KUKA KRL program: EPS_2_25694_GD05_A_20260114065905.src

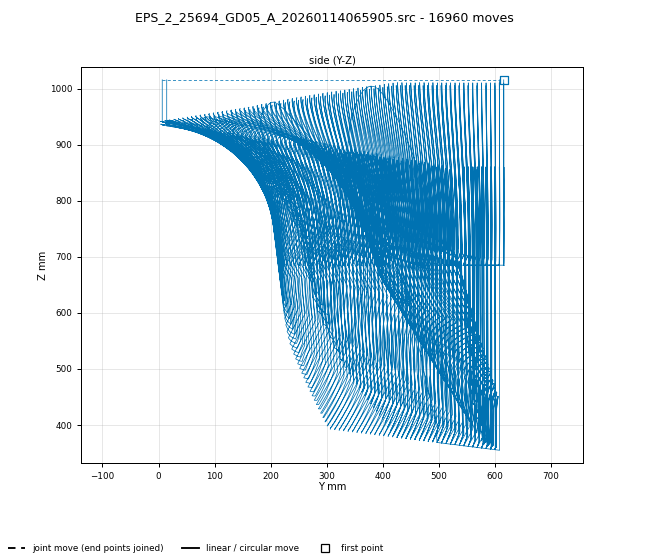
[picture p0: tool path of EPS_2_25694_GD05_A_20260114065905.src, 16960 of 16962 moves have a stored position in this frame; points joined in program order, loops and branches not executed]
&ACCESS RVP
&REL 4
&COMMENT QRS 19112012
&PARAM EDITMASK = *
DEF PART()
EXT BAS (BAS_COMMAND :IN,REAL :IN )
INT I
BAS (#INITMOV,0 )

;KUKA QRS Post kuka4.cps  Date:22-06-2017 !

File_ID=2971

QRS_PRE_INIT()

;Init var - Until changes are made in qrs_pre_init
Outlet_Square_prg=0
Inlet_1_Square_prg=0
Inlet_2_Square_prg=0
Inlet_3_Square_prg=0
Inlet_4_Square_prg=0
Inlet_5_Square_prg=0

Outlet_1={X 0.000, Y 425.000, Z 739.000, B 0.000, E1 0.000 }
Inlet_1={X 0.000, Y 500.470, Z 672.500, B 0.000, E1 180.000 }
Inlet_2={X 0.000, Y 520.810, Z 600.000, B 0.000, E1 270.000 }
Outlet_1_type=533
Inlet_1_type=366
Inlet_2_type=251
;QRS#1=Sidecore dimensions
;QRS#2=525-21" Concrete
;QRS#3=375-15" PVC SDR 35
;QRS#4=250-10" PVC SDR 35
;QRS#5=
;QRS#6=
;QRS#7=
;QRS#8=
;QRS#9=S306-32
;QRS#10=20Y PSX
;QRS#11=14M PSX
;QRS#12=
;QRS#13=
;QRS#14=
;QRS#15=
;QRS#16=1220x127x1372 4,5'
;QRS#17=EPS Height
;QRS#18=1005,5
;QRS#19=*
;QRS#20= UPDATED VERSION 22-06-2017
;QRS#21=*
Outlet_Square=0250
Inlet_1_Square=0250
Inlet_2_Square=0100
Inlet_3_Square=0
Inlet_4_Square=0
Inlet_5_Square=0
Mill_Square=1
Outlet_Square_Prg=263
Inlet_1_Square_prg=252
Inlet_2_Square_prg=205

QRS_INIT()

$ADVANCE=5

; T1
PTP {E1 172.561,E2 172.561}
PTP {X 0,Y 615.584,A -85,B 0,C 180,E1 172.561,E2 172.561,E3 0,E4 0,E5 0,E6 0}
QRS_SPEED_INIT()
LIN {X 0,Y 615.584,Z 1015.5,A -85,B 0,C 180,E1 172.561,E2 172.561,E3 0,E4 0,E5 0,E6 0} C_VEL
LIN {X 0,Y 615.584,Z 687.03,A -85,B 0,C 180,E1 172.561,E2 172.561} C_VEL
LIN {X 0,Y 615.53,Z 685.03,A -85,B 0,C 180,E1 172.747,E2 172.747} C_VEL
LIN {X 0,Y 615.824,Z 685.03,A -85,B 0,C 180,E1 176.52,E2 176.52} C_VEL
LIN {X 0,Y 615.876,Z 685.03,A -85,B 0,C 180,E1 181.159,E2 181.159} C_VEL
LIN {X 0,Y 615.817,Z 685.03,A -85,B 0,C 180,E1 185.807,E2 185.807} C_VEL
LIN {X 0,Y 615.791,Z 685.03,A -85,B 0,C 180,E1 190.494,E2 190.494} C_VEL
LIN {X 0,Y 615.808,Z 685.03,A -85,B 0,C 180,E1 195.252,E2 195.252} C_VEL
LIN {X 0,Y 615.745,Z 685.03,A -85,B 0,C 180,E1 200.123,E2 200.123} C_VEL
LIN {X 0,Y 615.743,Z 685.03,A -85,B 0,C 180,E1 205.15,E2 205.15} C_VEL
LIN {X 0,Y 615.401,Z 685.03,A -85,B 0,C 180,E1 209.459,E2 209.459} C_VEL
LIN {X 0,Y 615.733,Z 685.03,A -85,B 0,C 180,E1 210.395,E2 210.395} C_VEL
LIN {X 0,Y 615.144,Z 685.03,A -85,B 0,C 180,E1 213.844,E2 213.844} C_VEL
LIN {X 0,Y 615.689,Z 685.03,A -85,B 0,C 180,E1 215.941,E2 215.941} C_VEL
LIN {X 0,Y 615.421,Z 685.03,A -85,B 0,C 180,E1 217.844,E2 217.844} C_VEL
LIN {X 0,Y 615.368,Z 685.03,A -85,B 0,C 180,E1 218.885,E2 218.885} C_VEL
LIN {X 0,Y 615.634,Z 685.03,A -85,B 0,C 180,E1 221.502,E2 221.502} C_VEL
LIN {X 0,Y 615.674,Z 685.03,A -85,B 0,C 180,E1 225.105,E2 225.105} C_VEL
LIN {X 0,Y 615.272,Z 685.03,A -85,B 0,C 180,E1 228.536,E2 228.536} C_VEL
LIN {X 0,Y 615.659,Z 685.03,A -85,B 0,C 180,E1 231.137,E2 231.137} C_VEL
LIN {X 0,Y 615.631,Z 685.03,A -85,B 0,C 180,E1 236.089,E2 236.089} C_VEL
LIN {X 0,Y 615.749,Z 685.03,A -85,B 0,C 180,E1 236.879,E2 236.879} C_VEL
LIN {X 0,Y 615.824,Z 685.03,A -85,B 0,C 180,E1 240.42,E2 240.42} C_VEL
LIN {X 0,Y 615.203,Z 685.053,A -85,B 0,C 180,E1 240.571,E2 240.571} C_VEL
LIN {X 0,Y 615.421,Z 754.722,A -85,B 0,C 180,E1 241.502,E2 241.502} C_VEL
LIN {X 0,Y 615.517,Z 765.422,A -85,B 0,C 180,E1 241.682,E2 241.682} C_VEL
LIN {X 0,Y 615.533,Z 778.963,A -85,B 0,C 180,E1 241.97,E2 241.97} C_VEL
LIN {X 0,Y 615.511,Z 788.536,A -85,B 0,C 180,E1 242.211,E2 242.211} C_VEL
LIN {X 0,Y 615.673,Z 804.515,A -85,B 0,C 180,E1 242.705,E2 242.705} C_VEL
LIN {X 0,Y 615.632,Z 816.95,A -85,B 0,C 180,E1 243.151,E2 243.151} C_VEL
LIN {X 0,Y 615.564,Z 826.866,A -85,B 0,C 180,E1 243.554,E2 243.554} C_VEL
LIN {X 0,Y 615.704,Z 842.591,A -85,B 0,C 180,E1 244.286,E2 244.286} C_VEL
LIN {X 0,Y 615.691,Z 854.939,A -85,B 0,C 180,E1 244.935,E2 244.935} C_VEL
LIN {X 0,Y 615.678,Z 866.614,A -85,B 0,C 180,E1 245.617,E2 245.617} C_VEL
LIN {X 0,Y 615.714,Z 878.406,A -85,B 0,C 180,E1 246.379,E2 246.379} C_VEL
LIN {X 0,Y 615.719,Z 889.085,A -85,B 0,C 180,E1 247.135,E2 247.135} C_VEL
LIN {X 0,Y 615.705,Z 900.389,A -85,B 0,C 180,E1 248.011,E2 248.011} C_VEL
LIN {X 0,Y 615.703,Z 909.651,A -85,B 0,C 180,E1 248.791,E2 248.791} C_VEL
LIN {X 0,Y 615.752,Z 919.788,A -85,B 0,C 180,E1 249.723,E2 249.723} C_VEL
LIN {X 0,Y 615.721,Z 929.052,A -85,B 0,C 180,E1 250.646,E2 250.646} C_VEL
LIN {X 0,Y 615.678,Z 937.422,A -85,B 0,C 180,E1 251.549,E2 251.549} C_VEL
LIN {X 0,Y 615.759,Z 945.774,A -85,B 0,C 180,E1 252.531,E2 252.531} C_VEL
LIN {X 0,Y 615.711,Z 953.68,A -85,B 0,C 180,E1 253.541,E2 253.541} C_VEL
LIN {X 0,Y 615.577,Z 960.425,A -85,B 0,C 180,E1 254.472,E2 254.472} C_VEL
LIN {X 0,Y 615.67,Z 968.06,A -85,B 0,C 180,E1 255.644,E2 255.644} C_VEL
LIN {X 0,Y 615.808,Z 973.436,A -85,B 0,C 180,E1 256.543,E2 256.543} C_VEL
LIN {X 0,Y 615.572,Z 979.909,A -85,B 0,C 180,E1 257.728,E2 257.728} C_VEL
LIN {X 0,Y 615.608,Z 985.624,A -85,B 0,C 180,E1 258.913,E2 258.913} C_VEL
LIN {X 0,Y 615.819,Z 990.635,A -85,B 0,C 180,E1 260.096,E2 260.096} C_VEL
LIN {X 0,Y 615.602,Z 995.063,A -85,B 0,C 180,E1 261.268,E2 261.268} C_VEL
LIN {X 0,Y 615.662,Z 999.448,A -85,B 0,C 180,E1 262.653,E2 262.653} C_VEL
LIN {X 0,Y 615.802,Z 1002.362,A -85,B 0,C 180,E1 263.747,E2 263.747} C_VEL
LIN {X 0,Y 615.601,Z 1004.4,A -85,B 0,C 180,E1 264.657,E2 264.657} C_VEL
LIN {X 0,Y 615.536,Z 1006.161,A -85,B 0,C 180,E1 265.588,E2 265.588} C_VEL
LIN {X 0,Y 615.635,Z 1007.593,A -85,B 0,C 180,E1 266.519,E2 266.519} C_VEL
LIN {X 0,Y 615.7,Z 1009.056,A -85,B 0,C 180,E1 267.912,E2 267.912} C_VEL
LIN {X 0,Y 615.544,Z 1009.716,A -85,B 0,C 180,E1 268.84,E2 268.84} C_VEL
LIN {X 0,Y 615.842,Z 1009.659,A -85,B 0,C 180,E1 271.16,E2 271.16} C_VEL
LIN {X 0,Y 615.558,Z 1008.719,A -85,B 0,C 180,E1 272.553,E2 272.553} C_VEL
LIN {X 0,Y 615.598,Z 1006.935,A -85,B 0,C 180,E1 273.947,E2 273.947} C_VEL
LIN {X 0,Y 615.805,Z 1005.333,A -85,B 0,C 180,E1 274.876,E2 274.876} C_VEL
LIN {X 0,Y 615.605,Z 1002.404,A -85,B 0,C 180,E1 276.252,E2 276.252} C_VEL
LIN {X 0,Y 615.625,Z 999.258,A -85,B 0,C 180,E1 277.421,E2 277.421} C_VEL
LIN {X 0,Y 615.798,Z 995.032,A -85,B 0,C 180,E1 278.73,E2 278.73} C_VEL
LIN {X 0,Y 615.583,Z 990.668,A -85,B 0,C 180,E1 279.908,E2 279.908} C_VEL
LIN {X 0,Y 615.638,Z 985.619,A -85,B 0,C 180,E1 281.087,E2 281.087} C_VEL
LIN {X 0,Y 615.808,Z 979.88,A -85,B 0,C 180,E1 282.268,E2 282.268} C_VEL
LIN {X 0,Y 615.627,Z 973.452,A -85,B 0,C 180,E1 283.461,E2 283.461} C_VEL
LIN {X 0,Y 615.697,Z 966.191,A -85,B 0,C 180,E1 284.655,E2 284.655} C_VEL
LIN {X 0,Y 615.81,Z 960.633,A -85,B 0,C 180,E1 285.488,E2 285.488} C_VEL
LIN {X 0,Y 615.662,Z 951.196,A -85,B 0,C 180,E1 286.791,E2 286.791} C_VEL
LIN {X 0,Y 615.737,Z 942.603,A -85,B 0,C 180,E1 287.853,E2 287.853} C_VEL
LIN {X 0,Y 615.77,Z 934.408,A -85,B 0,C 180,E1 288.785,E2 288.785} C_VEL
LIN {X 0,Y 615.695,Z 924.518,A -85,B 0,C 180,E1 289.817,E2 289.817} C_VEL
LIN {X 0,Y 615.712,Z 916.531,A -85,B 0,C 180,E1 290.588,E2 290.588} C_VEL
LIN {X 0,Y 615.743,Z 906.028,A -85,B 0,C 180,E1 291.519,E2 291.519} C_VEL
LIN {X 0,Y 615.702,Z 896.055,A -85,B 0,C 180,E1 292.335,E2 292.335} C_VEL
LIN {X 0,Y 615.701,Z 886.287,A -85,B 0,C 180,E1 293.072,E2 293.072} C_VEL
LIN {X 0,Y 615.683,Z 874.63,A -85,B 0,C 180,E1 293.874,E2 293.874} C_VEL
LIN {X 0,Y 615.702,Z 862.594,A -85,B 0,C 180,E1 294.623,E2 294.623} C_VEL
LIN {X 0,Y 615.65,Z 851.876,A -85,B 0,C 180,E1 295.235,E2 295.235} C_VEL
LIN {X 0,Y 615.643,Z 841.007,A -85,B 0,C 180,E1 295.797,E2 295.797} C_VEL
LIN {X 0,Y 615.687,Z 826.859,A -85,B 0,C 180,E1 296.441,E2 296.441} C_VEL
LIN {X 0,Y 615.612,Z 813.654,A -85,B 0,C 180,E1 296.972,E2 296.972} C_VEL
LIN {X 0,Y 615.555,Z 804.507,A -85,B 0,C 180,E1 297.301,E2 297.301} C_VEL
LIN {X 0,Y 615.62,Z 787.838,A -85,B 0,C 180,E1 297.801,E2 297.801} C_VEL
LIN {X 0,Y 615.469,Z 776.068,A -85,B 0,C 180,E1 298.103,E2 298.103} C_VEL
LIN {X 0,Y 615.637,Z 761.901,A -85,B 0,C 180,E1 298.376,E2 298.376} C_VEL
LIN {X 0,Y 615.601,Z 741.63,A -85,B 0,C 180,E1 298.669,E2 298.669} C_VEL
LIN {X 0,Y 615.253,Z 685.03,A -85,B 0,C 180,E1 299.434,E2 299.434} C_VEL
LIN {X 0,Y 615.616,Z 685.03,A -85,B 0,C 180,E1 299.501,E2 299.501} C_VEL
LIN {X 0,Y 615.665,Z 685.03,A -85,B 0,C 180,E1 300.399,E2 300.399} C_VEL
LIN {X 0,Y 615.751,Z 685.03,A -85,B 0,C 180,E1 303.122,E2 303.122} C_VEL
LIN {X 0,Y 615.639,Z 685.03,A -85,B 0,C 180,E1 303.912,E2 303.912} C_VEL
LIN {X 0,Y 615.658,Z 685.03,A -85,B 0,C 180,E1 308.863,E2 308.863} C_VEL
LIN {X 0,Y 615.255,Z 685.03,A -85,B 0,C 180,E1 311.942,E2 311.942} C_VEL
LIN {X 0,Y 615.672,Z 685.03,A -85,B 0,C 180,E1 314.894,E2 314.894} C_VEL
LIN {X 0,Y 615.654,Z 685.03,A -85,B 0,C 180,E1 318.496,E2 318.496} C_VEL
LIN {X 0,Y 615.381,Z 685.03,A -85,B 0,C 180,E1 321.116,E2 321.116} C_VEL
LIN {X 0,Y 615.438,Z 685.03,A -85,B 0,C 180,E1 322.155,E2 322.155} C_VEL
LIN {X 0,Y 615.695,Z 685.03,A -85,B 0,C 180,E1 324.059,E2 324.059} C_VEL
LIN {X 0,Y 615.138,Z 685.03,A -85,B 0,C 180,E1 326.841,E2 326.841} C_VEL
LIN {X 0,Y 615.715,Z 685.03,A -85,B 0,C 180,E1 329.604,E2 329.604} C_VEL
LIN {X 0,Y 615.214,Z 685.03,A -85,B 0,C 180,E1 332.233,E2 332.233} C_VEL
LIN {X 0,Y 615.76,Z 685.03,A -85,B 0,C 180,E1 334.85,E2 334.85} C_VEL
LIN {X 0,Y 615.776,Z 685.03,A -85,B 0,C 180,E1 339.878,E2 339.878} C_VEL
LIN {X 0,Y 615.756,Z 685.03,A -85,B 0,C 180,E1 344.747,E2 344.747} C_VEL
LIN {X 0,Y 615.177,Z 685.03,A -85,B 0,C 180,E1 344.957,E2 344.957} C_VEL
LIN {X 0,Y 615.457,Z 685.827,A -85,B 0,C 180,E1 344.981,E2 344.981} C_VEL
LIN {X 0,Y 615.716,Z 687.593,A -85,B 0,C 180,E1 345.008,E2 345.008} C_VEL
LIN {X 0,Y 615.804,Z 728.118,A -85,B 0,C 180,E1 345.498,E2 345.498} C_VEL
LIN {X 0,Y 615.783,Z 737.858,A -85,B 0,C 180,E1 345.666,E2 345.666} C_VEL
LIN {X 0,Y 615.759,Z 747.806,A -85,B 0,C 180,E1 345.908,E2 345.908} C_VEL
LIN {X 0,Y 615.82,Z 756.4,A -85,B 0,C 180,E1 346.171,E2 346.171} C_VEL
LIN {X 0,Y 615.832,Z 766.418,A -85,B 0,C 180,E1 346.544,E2 346.544} C_VEL
LIN {X 0,Y 615.818,Z 774.745,A -85,B 0,C 180,E1 346.916,E2 346.916} C_VEL
LIN {X 0,Y 615.831,Z 783.402,A -85,B 0,C 180,E1 347.362,E2 347.362} C_VEL
LIN {X 0,Y 615.825,Z 792.017,A -85,B 0,C 180,E1 347.881,E2 347.881} C_VEL
LIN {X 0,Y 615.821,Z 799.559,A -85,B 0,C 180,E1 348.399,E2 348.399} C_VEL
LIN {X 0,Y 615.811,Z 808.029,A -85,B 0,C 180,E1 349.064,E2 349.064} C_VEL
LIN {X 0,Y 615.849,Z 814.611,A -85,B 0,C 180,E1 349.655,E2 349.655} C_VEL
LIN {X 0,Y 615.797,Z 821.882,A -85,B 0,C 180,E1 350.39,E2 350.39} C_VEL
LIN {X 0,Y 615.799,Z 828.194,A -85,B 0,C 180,E1 351.124,E2 351.124} C_VEL
LIN {X 0,Y 615.843,Z 833.772,A -85,B 0,C 180,E1 351.857,E2 351.857} C_VEL
LIN {X 0,Y 615.769,Z 838.545,A -85,B 0,C 180,E1 352.576,E2 352.576} C_VEL
LIN {X 0,Y 615.759,Z 842.466,A -85,B 0,C 180,E1 353.245,E2 353.245} C_VEL
LIN {X 0,Y 615.84,Z 847.264,A -85,B 0,C 180,E1 354.193,E2 354.193} C_VEL
LIN {X 0,Y 615.718,Z 851.122,A -85,B 0,C 180,E1 355.124,E2 355.124} C_VEL
LIN {X 0,Y 615.753,Z 854.265,A -85,B 0,C 180,E1 356.054,E2 356.054} C_VEL
LIN {X 0,Y 615.82,Z 856.63,A -85,B 0,C 180,E1 356.984,E2 356.984} C_VEL
LIN {X 0,Y 615.759,Z 857.615,A -85,B 0,C 180,E1 357.448,E2 357.448} C_VEL
LIN {X 0,Y 615.72,Z 858.999,A -85,B 0,C 180,E1 358.376,E2 358.376} C_VEL
LIN {X 0,Y 615.841,Z 859.769,A -85,B 0,C 180,E1 359.304,E2 359.304} C_VEL
LIN {X 0,Y 615.711,Z 859.892,A -85,B 0,C 180,E1 360.232,E2 360.232} C_VEL
LIN {X 0,Y 615.685,Z 859.413,A -85,B 0,C 180,E1 361.16,E2 361.16} C_VEL
LIN {X 0,Y 615.732,Z 858.891,A -85,B 0,C 180,E1 361.624,E2 361.624} C_VEL
LIN {X 0,Y 615.833,Z 857.437,A -85,B 0,C 180,E1 362.551,E2 362.551} C_VEL
LIN {X 0,Y 615.722,Z 855.292,A -85,B 0,C 180,E1 363.481,E2 363.481} C_VEL
LIN {X 0,Y 615.773,Z 852.487,A -85,B 0,C 180,E1 364.41,E2 364.41} C_VEL
LIN {X 0,Y 615.847,Z 850.762,A -85,B 0,C 180,E1 364.875,E2 364.875} C_VEL
LIN {X 0,Y 615.751,Z 846.849,A -85,B 0,C 180,E1 365.808,E2 365.808} C_VEL
LIN {X 0,Y 615.738,Z 841.761,A -85,B 0,C 180,E1 366.794,E2 366.794} C_VEL
LIN {X 0,Y 615.85,Z 836.822,A -85,B 0,C 180,E1 367.602,E2 367.602} C_VEL
LIN {X 0,Y 615.766,Z 830.942,A -85,B 0,C 180,E1 368.437,E2 368.437} C_VEL
LIN {X 0,Y 615.764,Z 825.022,A -85,B 0,C 180,E1 369.17,E2 369.17} C_VEL
LIN {X 0,Y 615.833,Z 819.636,A -85,B 0,C 180,E1 369.757,E2 369.757} C_VEL
LIN {X 0,Y 615.834,Z 813.655,A -85,B 0,C 180,E1 370.346,E2 370.346} C_VEL
LIN {X 0,Y 615.806,Z 806.983,A -85,B 0,C 180,E1 370.936,E2 370.936} C_VEL
LIN {X 0,Y 615.829,Z 799.335,A -85,B 0,C 180,E1 371.527,E2 371.527} C_VEL
LIN {X 0,Y 615.844,Z 791.773,A -85,B 0,C 180,E1 372.044,E2 372.044} C_VEL
LIN {X 0,Y 615.819,Z 783.109,A -85,B 0,C 180,E1 372.564,E2 372.564} C_VEL
LIN {X 0,Y 615.806,Z 774.421,A -85,B 0,C 180,E1 373.01,E2 373.01} C_VEL
LIN {X 0,Y 615.823,Z 766.055,A -85,B 0,C 180,E1 373.382,E2 373.382} C_VEL
LIN {X 0,Y 615.826,Z 755.927,A -85,B 0,C 180,E1 373.755,E2 373.755} C_VEL
LIN {X 0,Y 615.788,Z 747.254,A -85,B 0,C 180,E1 374.017,E2 374.017} C_VEL
LIN {X 0,Y 615.813,Z 739.659,A -85,B 0,C 180,E1 374.203,E2 374.203} C_VEL
LIN {X 0,Y 615.835,Z 729.706,A -85,B 0,C 180,E1 374.389,E2 374.389} C_VEL
LIN {X 0,Y 615.679,Z 699.013,A -85,B 0,C 180,E1 374.768,E2 374.768} C_VEL
LIN {X 0,Y 615.543,Z 686.33,A -85,B 0,C 180,E1 374.921,E2 374.921} C_VEL
LIN {X 0,Y 615.607,Z 685.03,A -85,B 0,C 180,E1 374.957,E2 374.957} C_VEL
LIN {X 0,Y 615.792,Z 685.03,A -85,B 0,C 180,E1 375.252,E2 375.252} C_VEL
LIN {X 0,Y 615.768,Z 685.03,A -85,B 0,C 180,E1 380.123,E2 380.123} C_VEL
LIN {X 0,Y 615.761,Z 685.03,A -85,B 0,C 180,E1 385.15,E2 385.15} C_VEL
LIN {X 0,Y 615.378,Z 685.03,A -85,B 0,C 180,E1 389.454,E2 389.454} C_VEL
LIN {X 0,Y 615.701,Z 685.03,A -85,B 0,C 180,E1 390.397,E2 390.397} C_VEL
LIN {X 0,Y 615.132,Z 685.03,A -85,B 0,C 180,E1 393.842,E2 393.842} C_VEL
LIN {X 0,Y 615.69,Z 685.03,A -85,B 0,C 180,E1 395.941,E2 395.941} C_VEL
LIN {X 0,Y 615.638,Z 685.03,A -85,B 0,C 180,E1 397.869,E2 397.869} C_VEL
LIN {X 0,Y 615.724,Z 685.03,A -85,B 0,C 180,E1 398.858,E2 398.858} C_VEL
LIN {X 0,Y 615.234,Z 685.03,A -85,B 0,C 180,E1 401.944,E2 401.944} C_VEL
LIN {X 0,Y 615.676,Z 685.03,A -85,B 0,C 180,E1 404.895,E2 404.895} C_VEL
LIN {X 0,Y 615.651,Z 685.03,A -85,B 0,C 180,E1 408.497,E2 408.497} C_VEL
LIN {X 0,Y 615.347,Z 685.03,A -85,B 0,C 180,E1 411.113,E2 411.113} C_VEL
LIN {X 0,Y 615.387,Z 685.03,A -85,B 0,C 180,E1 412.161,E2 412.161} C_VEL
LIN {X 0,Y 615.636,Z 685.03,A -85,B 0,C 180,E1 414.055,E2 414.055} C_VEL
LIN {X 0,Y 615.128,Z 685.03,A -85,B 0,C 180,E1 416.84,E2 416.84} C_VEL
LIN {X 0,Y 615.747,Z 685.03,A -85,B 0,C 180,E1 419.606,E2 419.606} C_VEL
LIN {X 0,Y 615.236,Z 685.03,A -85,B 0,C 180,E1 422.234,E2 422.234} C_VEL
LIN {X 0,Y 615.77,Z 685.03,A -85,B 0,C 180,E1 424.851,E2 424.851} C_VEL
LIN {X 0,Y 615.275,Z 685.03,A -85,B 0,C 180,E1 427.368,E2 427.368} C_VEL
LIN {X 0,Y 615.552,Z 685.03,A -85,B 0,C 180,E1 429.87,E2 429.87} C_VEL
LIN {X 0,Y 614.862,Z 685.03,A -85,B 0,C 180,E1 430.001,E2 430.001} C_VEL
LIN {X 0,Y 615.158,Z 686.38,A -85,B 0,C 180,E1 430.056,E2 430.056} C_VEL
LIN {X 0,Y 615.519,Z 688.076,A -85,B 0,C 180,E1 430.1,E2 430.1} C_VEL
LIN {X 0,Y 615.754,Z 695.441,A -85,B 0,C 180,E1 430.262,E2 430.262} C_VEL
LIN {X 0,Y 615.807,Z 705.296,A -85,B 0,C 180,E1 430.514,E2 430.514} C_VEL
LIN {X 0,Y 615.785,Z 714.797,A -85,B 0,C 180,E1 430.801,E2 430.801} C_VEL
LIN {X 0,Y 615.726,Z 723.53,A -85,B 0,C 180,E1 431.106,E2 431.106} C_VEL
LIN {X 0,Y 615.788,Z 732.709,A -85,B 0,C 180,E1 431.477,E2 431.477} C_VEL
LIN {X 0,Y 615.779,Z 741.924,A -85,B 0,C 180,E1 431.897,E2 431.897} C_VEL
LIN {X 0,Y 615.726,Z 750.371,A -85,B 0,C 180,E1 432.327,E2 432.327} C_VEL
LIN {X 0,Y 615.768,Z 758.249,A -85,B 0,C 180,E1 432.773,E2 432.773} C_VEL
LIN {X 0,Y 615.772,Z 765.444,A -85,B 0,C 180,E1 433.217,E2 433.217} C_VEL
LIN {X 0,Y 615.802,Z 774.115,A -85,B 0,C 180,E1 433.81,E2 433.81} C_VEL
LIN {X 0,Y 615.788,Z 781.849,A -85,B 0,C 180,E1 434.39,E2 434.39} C_VEL
LIN {X 0,Y 615.765,Z 789.814,A -85,B 0,C 180,E1 435.047,E2 435.047} C_VEL
LIN {X 0,Y 615.775,Z 796.45,A -85,B 0,C 180,E1 435.647,E2 435.647} C_VEL
LIN {X 0,Y 615.829,Z 803.981,A -85,B 0,C 180,E1 436.395,E2 436.395} C_VEL
LIN {X 0,Y 615.772,Z 809.484,A -85,B 0,C 180,E1 436.989,E2 436.989} C_VEL
LIN {X 0,Y 615.717,Z 815.784,A -85,B 0,C 180,E1 437.731,E2 437.731} C_VEL
LIN {X 0,Y 615.762,Z 821.496,A -85,B 0,C 180,E1 438.472,E2 438.472} C_VEL
LIN {X 0,Y 615.83,Z 826.677,A -85,B 0,C 180,E1 439.212,E2 439.212} C_VEL
LIN {X 0,Y 615.701,Z 832.297,A -85,B 0,C 180,E1 440.094,E2 440.094} C_VEL
LIN {X 0,Y 615.677,Z 835.681,A -85,B 0,C 180,E1 440.681,E2 440.681} C_VEL
LIN {X 0,Y 615.761,Z 840.253,A -85,B 0,C 180,E1 441.563,E2 441.563} C_VEL
LIN {X 0,Y 615.825,Z 843.092,A -85,B 0,C 180,E1 442.165,E2 442.165} C_VEL
LIN {X 0,Y 615.696,Z 846.093,A -85,B 0,C 180,E1 442.859,E2 442.859} C_VEL
LIN {X 0,Y 615.628,Z 849.335,A -85,B 0,C 180,E1 443.719,E2 443.719} C_VEL
LIN {X 0,Y 615.712,Z 852.329,A -85,B 0,C 180,E1 444.658,E2 444.658} C_VEL
LIN {X 0,Y 615.79,Z 854.78,A -85,B 0,C 180,E1 445.59,E2 445.59} C_VEL
LIN {X 0,Y 615.639,Z 856.773,A -85,B 0,C 180,E1 446.519,E2 446.519} C_VEL
LIN {X 0,Y 615.653,Z 858.252,A -85,B 0,C 180,E1 447.448,E2 447.448} C_VEL
LIN {X 0,Y 615.775,Z 859.568,A -85,B 0,C 180,E1 448.84,E2 448.84} C_VEL
LIN {X 0,Y 615.634,Z 859.928,A -85,B 0,C 180,E1 449.768,E2 449.768} C_VEL
LIN {X 0,Y 615.624,Z 859.908,A -85,B 0,C 180,E1 450.232,E2 450.232} C_VEL
LIN {X 0,Y 615.725,Z 859.514,A -85,B 0,C 180,E1 451.16,E2 451.16} C_VEL
LIN {X 0,Y 615.786,Z 858.668,A -85,B 0,C 180,E1 452.087,E2 452.087} C_VEL
LIN {X 0,Y 615.702,Z 858.137,A -85,B 0,C 180,E1 452.552,E2 452.552} C_VEL
LIN {X 0,Y 615.627,Z 856.622,A -85,B 0,C 180,E1 453.481,E2 453.481} C_VEL
LIN {X 0,Y 615.721,Z 854.584,A -85,B 0,C 180,E1 454.411,E2 454.411} C_VEL
LIN {X 0,Y 615.769,Z 852.048,A -85,B 0,C 180,E1 455.341,E2 455.341} C_VEL
LIN {X 0,Y 615.671,Z 848.986,A -85,B 0,C 180,E1 456.283,E2 456.283} C_VEL
LIN {X 0,Y 615.764,Z 844.496,A -85,B 0,C 180,E1 457.42,E2 457.42} C_VEL
LIN {X 0,Y 615.808,Z 841.234,A -85,B 0,C 180,E1 458.143,E2 458.143} C_VEL
LIN {X 0,Y 615.717,Z 838.386,A -85,B 0,C 180,E1 458.731,E2 458.731} C_VEL
LIN {X 0,Y 615.682,Z 833.542,A -85,B 0,C 180,E1 459.612,E2 459.612} C_VEL
LIN {X 0,Y 615.79,Z 828.06,A -85,B 0,C 180,E1 460.494,E2 460.494} C_VEL
LIN {X 0,Y 615.811,Z 823.014,A -85,B 0,C 180,E1 461.231,E2 461.231} C_VEL
LIN {X 0,Y 615.725,Z 817.46,A -85,B 0,C 180,E1 461.972,E2 461.972} C_VEL
LIN {X 0,Y 615.74,Z 811.326,A -85,B 0,C 180,E1 462.714,E2 462.714} C_VEL
LIN {X 0,Y 615.83,Z 804.554,A -85,B 0,C 180,E1 463.456,E2 463.456} C_VEL
LIN {X 0,Y 615.807,Z 798.651,A -85,B 0,C 180,E1 464.053,E2 464.053} C_VEL
LIN {X 0,Y 615.764,Z 792.222,A -85,B 0,C 180,E1 464.653,E2 464.653} C_VEL
LIN {X 0,Y 615.786,Z 785.195,A -85,B 0,C 180,E1 465.252,E2 465.252} C_VEL
LIN {X 0,Y 615.795,Z 777.438,A -85,B 0,C 180,E1 465.857,E2 465.857} C_VEL
LIN {X 0,Y 615.796,Z 770.063,A -85,B 0,C 180,E1 466.384,E2 466.384} C_VEL
LIN {X 0,Y 615.768,Z 762.769,A -85,B 0,C 180,E1 466.863,E2 466.863} C_VEL
LIN {X 0,Y 615.76,Z 754.276,A -85,B 0,C 180,E1 467.368,E2 467.368} C_VEL
LIN {X 0,Y 615.734,Z 744.638,A -85,B 0,C 180,E1 467.881,E2 467.881} C_VEL
LIN {X 0,Y 615.774,Z 735.788,A -85,B 0,C 180,E1 468.299,E2 468.299} C_VEL
LIN {X 0,Y 615.768,Z 726.909,A -85,B 0,C 180,E1 468.672,E2 468.672} C_VEL
LIN {X 0,Y 615.7,Z 718.531,A -85,B 0,C 180,E1 468.987,E2 468.987} C_VEL
LIN {X 0,Y 615.806,Z 708.175,A -85,B 0,C 180,E1 469.314,E2 469.314} C_VEL
LIN {X 0,Y 615.799,Z 698.822,A -85,B 0,C 180,E1 469.566,E2 469.566} C_VEL
LIN {X 0,Y 615.703,Z 688.908,A -85,B 0,C 180,E1 469.788,E2 469.788} C_VEL
LIN {X 0,Y 615.636,Z 685.03,A -85,B 0,C 180,E1 469.874,E2 469.874} C_VEL
LIN {X 0,Y 615.853,Z 685.03,A -85,B 0,C 180,E1 469.985,E2 469.985} C_VEL
LIN {X 0,Y 615.83,Z 685.03,A -85,B 0,C 180,E1 472.61,E2 472.61} C_VEL
LIN {X 0,Y 615.75,Z 685.03,A -85,B 0,C 180,E1 477.74,E2 477.74} C_VEL
LIN {X 0,Y 615.174,Z 685.03,A -85,B 0,C 180,E1 480.425,E2 480.425} C_VEL
LIN {X 0,Y 615.698,Z 685.03,A -85,B 0,C 180,E1 483.125,E2 483.125} C_VEL
LIN {X 0,Y 615.634,Z 685.03,A -85,B 0,C 180,E1 483.911,E2 483.911} C_VEL
LIN {X 0,Y 615.656,Z 685.03,A -85,B 0,C 180,E1 488.863,E2 488.863} C_VEL
LIN {X 0,Y 615.247,Z 685.03,A -85,B 0,C 180,E1 491.943,E2 491.943} C_VEL
LIN {X 0,Y 615.653,Z 685.03,A -85,B 0,C 180,E1 494.893,E2 494.893} C_VEL
LIN {X 0,Y 615.627,Z 685.03,A -85,B 0,C 180,E1 498.499,E2 498.499} C_VEL
LIN {X 0,Y 615.365,Z 685.03,A -85,B 0,C 180,E1 501.115,E2 501.115} C_VEL
LIN {X 0,Y 615.417,Z 685.03,A -85,B 0,C 180,E1 502.157,E2 502.157} C_VEL
LIN {X 0,Y 615.697,Z 685.03,A -85,B 0,C 180,E1 504.06,E2 504.06} C_VEL
LIN {X 0,Y 615.157,Z 685.03,A -85,B 0,C 180,E1 506.842,E2 506.842} C_VEL
LIN {X 0,Y 615.745,Z 685.03,A -85,B 0,C 180,E1 509.606,E2 509.606} C_VEL
LIN {X 0,Y 615.215,Z 685.03,A -85,B 0,C 180,E1 512.233,E2 512.233} C_VEL
LIN {X 0,Y 615.723,Z 685.03,A -85,B 0,C 180,E1 514.849,E2 514.849} C_VEL
LIN {X 0,Y 615.778,Z 685.03,A -85,B 0,C 180,E1 519.878,E2 519.878} C_VEL
LIN {X 0,Y 615.515,Z 685.03,A -85,B 0,C 180,E1 522.321,E2 522.321} C_VEL
LIN {X 0,Y 615.64,Z 685.03,A -85,B 0,C 180,E1 524.744,E2 524.744} C_VEL
LIN {X 0,Y 615.831,Z 685.03,A -85,B 0,C 180,E1 527.139,E2 527.139} C_VEL
LIN {X 0,Y 615.834,Z 685.03,A -85,B 0,C 180,E1 531.857,E2 531.857} C_VEL
LIN {X 0,Y 615.53,Z 685.03,A -85,B 0,C 180,E1 532.747,E2 532.747} C_VEL
LIN {X 0,Y 611.514,Z 685.03,A -85,B 0,C 180,E1 534.334,E2 534.334} C_VEL
LIN {X 0,Y 607.65,Z 685.03,A -85,B 0,C 180,E1 535.941,E2 535.941} C_VEL
LIN {X 0,Y 607.884,Z 685.03,A -85,B 0,C 180,E1 541.425,E2 541.425} C_VEL
LIN {X 0,Y 607.635,Z 685.03,A -85,B 0,C 180,E1 546.599,E2 546.599} C_VEL
LIN {X 0,Y 607.552,Z 685.03,A -85,B 0,C 180,E1 551.463,E2 551.463} C_VEL
LIN {X 0,Y 607.655,Z 685.03,A -85,B 0,C 180,E1 555.855,E2 555.855} C_VEL
LIN {X 0,Y 607.757,Z 685.03,A -85,B 0,C 180,E1 560.343,E2 560.343} C_VEL
LIN {X 0,Y 607.766,Z 685.03,A -85,B 0,C 180,E1 564.968,E2 564.968} C_VEL
LIN {X 0,Y 607.612,Z 685.03,A -85,B 0,C 180,E1 569.783,E2 569.783} C_VEL
LIN {X 0,Y 607.625,Z 685.03,A -85,B 0,C 180,E1 576.586,E2 576.586} C_VEL
LIN {X 0,Y 607.595,Z 685.03,A -85,B 0,C 180,E1 582.11,E2 582.11} C_VEL
LIN {X 0,Y 607.278,Z 685.03,A -85,B 0,C 180,E1 587.863,E2 587.863} C_VEL
LIN {X 0,Y 607.283,Z 685.03,A -85,B 0,C 180,E1 592.668,E2 592.668} C_VEL
LIN {X 0,Y 607.689,Z 685.03,A -85,B 0,C 180,E1 597.593,E2 597.593} C_VEL
LIN {X 0,Y 607.848,Z 685.03,A -85,B 0,C 180,E1 600.149,E2 600.149} C_VEL
LIN {X 0,Y 608.576,Z 775.688,A -85,B 0,C 180,E1 601.541,E2 601.541} C_VEL
LIN {X 0,Y 608.525,Z 816.222,A -85,B 0,C 180,E1 602.783,E2 602.783} C_VEL
LIN {X 0,Y 608.423,Z 854.222,A -85,B 0,C 180,E1 604.573,E2 604.573} C_VEL
LIN {X 0,Y 608.249,Z 889.948,A -85,B 0,C 180,E1 606.904,E2 606.904} C_VEL
LIN {X 0,Y 608.103,Z 921.971,A -85,B 0,C 180,E1 609.672,E2 609.672} C_VEL
LIN {X 0,Y 607.995,Z 948.714,A -85,B 0,C 180,E1 612.674,E2 612.674} C_VEL
LIN {X 0,Y 607.894,Z 971.358,A -85,B 0,C 180,E1 615.995,E2 615.995} C_VEL
LIN {X 0,Y 607.873,Z 989.524,A -85,B 0,C 180,E1 619.633,E2 619.633} C_VEL
LIN {X 0,Y 607.904,Z 1002.409,A -85,B 0,C 180,E1 623.517,E2 623.517} C_VEL
LIN {X 0,Y 607.762,Z 1008.909,A -85,B 0,C 180,E1 627.156,E2 627.156} C_VEL
LIN {X 0,Y 607.732,Z 1010.5,A -85,B 0,C 180,E1 630.002,E2 630.002} C_VEL
LIN {X 0,Y 607.681,Z 1008.904,A -85,B 0,C 180,E1 632.849,E2 632.849} C_VEL
LIN {X 0,Y 607.746,Z 1002.587,A -85,B 0,C 180,E1 636.418,E2 636.418} C_VEL
LIN {X 0,Y 607.726,Z 991.034,A -85,B 0,C 180,E1 640.012,E2 640.012} C_VEL
LIN {X 0,Y 607.791,Z 973.516,A -85,B 0,C 180,E1 643.645,E2 643.645} C_VEL
LIN {X 0,Y 607.899,Z 951.608,A -85,B 0,C 180,E1 646.961,E2 646.961} C_VEL
LIN {X 0,Y 608.055,Z 924.838,A -85,B 0,C 180,E1 650.045,E2 650.045} C_VEL
LIN {X 0,Y 608.197,Z 893.631,A -85,B 0,C 180,E1 652.813,E2 652.813} C_VEL
LIN {X 0,Y 608.356,Z 859.179,A -85,B 0,C 180,E1 655.14,E2 655.14} C_VEL
LIN {X 0,Y 608.506,Z 823.626,A -85,B 0,C 180,E1 656.912,E2 656.912} C_VEL
LIN {X 0,Y 608.583,Z 787.466,A -85,B 0,C 180,E1 658.161,E2 658.161} C_VEL
LIN {X 0,Y 608.697,Z 746.264,A -85,B 0,C 180,E1 658.964,E2 658.964} C_VEL
LIN {X 0,Y 607.721,Z 685.15,A -85,B 0,C 180,E1 659.827,E2 659.827} C_VEL
LIN {X 0,Y 607.861,Z 685.03,A -85,B 0,C 180,E1 663.107,E2 663.107} C_VEL
LIN {X 0,Y 607.486,Z 685.03,A -85,B 0,C 180,E1 669.643,E2 669.643} C_VEL
LIN {X 0,Y 607.532,Z 685.03,A -85,B 0,C 180,E1 675.936,E2 675.936} C_VEL
LIN {X 0,Y 607.454,Z 685.03,A -85,B 0,C 180,E1 680.368,E2 680.368} C_VEL
LIN {X 0,Y 607.426,Z 685.03,A -85,B 0,C 180,E1 685.153,E2 685.153} C_VEL
LIN {X 0,Y 607.533,Z 685.03,A -85,B 0,C 180,E1 690.391,E2 690.391} C_VEL
LIN {X 0,Y 607.798,Z 685.03,A -85,B 0,C 180,E1 695.034,E2 695.034} C_VEL
LIN {X 0,Y 607.557,Z 685.03,A -85,B 0,C 180,E1 700.717,E2 700.717} C_VEL
LIN {X 0,Y 607.618,Z 685.03,A -85,B 0,C 180,E1 704.74,E2 704.74} C_VEL
LIN {X 0,Y 608.135,Z 742.995,A -85,B 0,C 180,E1 705.602,E2 705.602} C_VEL
LIN {X 0,Y 608.142,Z 770.479,A -85,B 0,C 180,E1 706.546,E2 706.546} C_VEL
LIN {X 0,Y 608.05,Z 796.203,A -85,B 0,C 180,E1 708.002,E2 708.002} C_VEL
LIN {X 0,Y 608.01,Z 819.489,A -85,B 0,C 180,E1 709.993,E2 709.993} C_VEL
LIN {X 0,Y 607.966,Z 836.748,A -85,B 0,C 180,E1 712.151,E2 712.151} C_VEL
LIN {X 0,Y 607.906,Z 849.994,A -85,B 0,C 180,E1 714.656,E2 714.656} C_VEL
LIN {X 0,Y 607.94,Z 857.604,A -85,B 0,C 180,E1 717.152,E2 717.152} C_VEL
LIN {X 0,Y 607.859,Z 860.496,A -85,B 0,C 180,E1 719.997,E2 719.997} C_VEL
LIN {X 0,Y 607.927,Z 857.423,A -85,B 0,C 180,E1 722.842,E2 722.842} C_VEL
LIN {X 0,Y 607.926,Z 849.636,A -85,B 0,C 180,E1 725.337,E2 725.337} C_VEL
LIN {X 0,Y 607.973,Z 836.187,A -85,B 0,C 180,E1 727.842,E2 727.842} C_VEL
LIN {X 0,Y 608.018,Z 816.927,A -85,B 0,C 180,E1 730.181,E2 730.181} C_VEL
LIN {X 0,Y 608.067,Z 793.615,A -85,B 0,C 180,E1 732.082,E2 732.082} C_VEL
LIN {X 0,Y 608.14,Z 766.434,A -85,B 0,C 180,E1 733.539,E2 733.539} C_VEL
LIN {X 0,Y 608.191,Z 737.961,A -85,B 0,C 180,E1 734.424,E2 734.424} C_VEL
LIN {X 0,Y 607.821,Z 685.03,A -85,B 0,C 180,E1 735.149,E2 735.149} C_VEL
LIN {X 0,Y 607.777,Z 685.03,A -85,B 0,C 180,E1 740.335,E2 740.335} C_VEL
LIN {X 0,Y 607.795,Z 685.03,A -85,B 0,C 180,E1 744.959,E2 744.959} C_VEL
LIN {X 0,Y 607.594,Z 685.03,A -85,B 0,C 180,E1 749.776,E2 749.776} C_VEL
LIN {X 0,Y 607.716,Z 685.03,A -85,B 0,C 180,E1 756.572,E2 756.572} C_VEL
LIN {X 0,Y 607.329,Z 685.03,A -85,B 0,C 180,E1 761.8,E2 761.8} C_VEL
LIN {X 0,Y 607.5,Z 685.03,A -85,B 0,C 180,E1 766.073,E2 766.073} C_VEL
LIN {X 0,Y 607.404,Z 685.03,A -85,B 0,C 180,E1 770.356,E2 770.356} C_VEL
LIN {X 0,Y 607.386,Z 685.03,A -85,B 0,C 180,E1 775.146,E2 775.146} C_VEL
LIN {X 0,Y 607.585,Z 685.03,A -85,B 0,C 180,E1 780.358,E2 780.358} C_VEL
LIN {X 0,Y 607.812,Z 685.03,A -85,B 0,C 180,E1 785.032,E2 785.032} C_VEL
LIN {X 0,Y 607.44,Z 685.03,A -85,B 0,C 180,E1 789.748,E2 789.748} C_VEL
LIN {X 0,Y 608.265,Z 720.247,A -85,B 0,C 180,E1 790.741,E2 790.741} C_VEL
LIN {X 0,Y 608.115,Z 752.314,A -85,B 0,C 180,E1 792.207,E2 792.207} C_VEL
LIN {X 0,Y 608.102,Z 781.459,A -85,B 0,C 180,E1 794.156,E2 794.156} C_VEL
LIN {X 0,Y 608.037,Z 807.114,A -85,B 0,C 180,E1 796.543,E2 796.543} C_VEL
LIN {X 0,Y 607.974,Z 828.18,A -85,B 0,C 180,E1 799.269,E2 799.269} C_VEL
LIN {X 0,Y 607.957,Z 843.82,A -85,B 0,C 180,E1 802.151,E2 802.151} C_VEL
LIN {X 0,Y 607.861,Z 853.912,A -85,B 0,C 180,E1 805.013,E2 805.013} C_VEL
LIN {X 0,Y 607.779,Z 858.393,A -85,B 0,C 180,E1 807.151,E2 807.151} C_VEL
LIN {X 0,Y 607.753,Z 860.497,A -85,B 0,C 180,E1 809.998,E2 809.998} C_VEL
LIN {X 0,Y 607.807,Z 858.251,A -85,B 0,C 180,E1 812.844,E2 812.844} C_VEL
LIN {X 0,Y 607.841,Z 850.443,A -85,B 0,C 180,E1 816.055,E2 816.055} C_VEL
LIN {X 0,Y 607.844,Z 838.233,A -85,B 0,C 180,E1 818.924,E2 818.924} C_VEL
LIN {X 0,Y 607.934,Z 819.971,A -85,B 0,C 180,E1 821.815,E2 821.815} C_VEL
LIN {X 0,Y 608.014,Z 796.178,A -85,B 0,C 180,E1 824.478,E2 824.478} C_VEL
LIN {X 0,Y 608.129,Z 768.961,A -85,B 0,C 180,E1 826.672,E2 826.672} C_VEL
LIN {X 0,Y 608.243,Z 737.927,A -85,B 0,C 180,E1 828.439,E2 828.439} C_VEL
LIN {X 0,Y 608.343,Z 705.223,A -85,B 0,C 180,E1 829.647,E2 829.647} C_VEL
LIN {X 0,Y 607.914,Z 685.03,A -85,B 0,C 180,E1 830.147,E2 830.147} C_VEL
LIN {X 0,Y 607.297,Z 685.03,A -85,B 0,C 180,E1 834.986,E2 834.986} C_VEL
LIN {X 0,Y 607.316,Z 685.03,A -85,B 0,C 180,E1 839.598,E2 839.598} C_VEL
LIN {X 0,Y 607.796,Z 685.03,A -85,B 0,C 180,E1 843.106,E2 843.106} C_VEL
LIN {X 0,Y 607.5,Z 685.03,A -85,B 0,C 180,E1 849.655,E2 849.655} C_VEL
LIN {X 0,Y 607.496,Z 685.03,A -85,B 0,C 180,E1 855.941,E2 855.941} C_VEL
LIN {X 0,Y 607.41,Z 685.03,A -85,B 0,C 180,E1 860.367,E2 860.367} C_VEL
LIN {X 0,Y 607.426,Z 685.03,A -85,B 0,C 180,E1 865.161,E2 865.161} C_VEL
LIN {X 0,Y 607.552,Z 685.03,A -85,B 0,C 180,E1 870.379,E2 870.379} C_VEL
LIN {X 0,Y 607.746,Z 685.03,A -85,B 0,C 180,E1 875.038,E2 875.038} C_VEL
LIN {X 0,Y 607.613,Z 685.03,A -85,B 0,C 180,E1 881.169,E2 881.169} C_VEL
LIN {X 0,Y 607.934,Z 685.03,A -85,B 0,C 180,E1 887.096,E2 887.096} C_VEL
LIN {X 0,Y 607.609,Z 685.03,A -85,B 0,C 180,E1 892.871,E2 892.871} C_VEL
LIN {X 0,Y 607.65,Z 685.03,A -85,B 0,C 180,E1 895.941,E2 895.941} C_VEL
LIN {X 0,Y 606.327,Z 685.03,A -85,B 0,C 180,E1 896.755,E2 896.755} C_VEL
LIN {X 0,Y 599.651,Z 685.03,A -85,B 0,C 180,E1 898.966,E2 898.966} C_VEL
LIN {X 0,Y 599.575,Z 685.03,A -85,B 0,C 180,E1 899.175,E2 899.175} C_VEL
LIN {X 0,Y 599.626,Z 685.03,A -85,B 0,C 180,E1 902.888,E2 902.888} C_VEL
LIN {X 0,Y 599.588,Z 685.03,A -85,B 0,C 180,E1 907.232,E2 907.232} C_VEL
LIN {X 0,Y 599.617,Z 685.03,A -85,B 0,C 180,E1 911.617,E2 911.617} C_VEL
LIN {X 0,Y 599.684,Z 685.03,A -85,B 0,C 180,E1 916.071,E2 916.071} C_VEL
LIN {X 0,Y 599.535,Z 685.03,A -85,B 0,C 180,E1 921.364,E2 921.364} C_VEL
LIN {X 0,Y 599.746,Z 685.03,A -85,B 0,C 180,E1 925.325,E2 925.325} C_VEL
LIN {X 0,Y 599.526,Z 685.03,A -85,B 0,C 180,E1 931.154,E2 931.154} C_VEL
LIN {X 0,Y 599.656,Z 685.03,A -85,B 0,C 180,E1 937.153,E2 937.153} C_VEL
LIN {X 0,Y 599.569,Z 685.03,A -85,B 0,C 180,E1 943.124,E2 943.124} C_VEL
LIN {X 0,Y 599.421,Z 685.03,A -85,B 0,C 180,E1 949.116,E2 949.116} C_VEL
LIN {X 0,Y 599.296,Z 685.03,A -85,B 0,C 180,E1 953.681,E2 953.681} C_VEL
LIN {X 0,Y 599.74,Z 685.03,A -85,B 0,C 180,E1 958.105,E2 958.105} C_VEL
LIN {X 0,Y 599.877,Z 685.425,A -85,B 0,C 180,E1 959.746,E2 959.746} C_VEL
LIN {X 0,Y 601.496,Z 692.445,A -85,B 0,C 180,E1 959.931,E2 959.931} C_VEL
LIN {X 0,Y 601.613,Z 773.311,A -85,B 0,C 180,E1 961.131,E2 961.131} C_VEL
LIN {X 0,Y 601.454,Z 811.075,A -85,B 0,C 180,E1 962.244,E2 962.244} C_VEL
LIN {X 0,Y 601.186,Z 846.851,A -85,B 0,C 180,E1 963.845,E2 963.845} C_VEL
LIN {X 0,Y 600.85,Z 881.964,A -85,B 0,C 180,E1 966.013,E2 966.013} C_VEL
LIN {X 0,Y 600.536,Z 913.084,A -85,B 0,C 180,E1 968.546,E2 968.546} C_VEL
LIN {X 0,Y 600.234,Z 941.137,A -85,B 0,C 180,E1 971.496,E2 971.496} C_VEL
LIN {X 0,Y 599.99,Z 965.765,A -85,B 0,C 180,E1 974.876,E2 974.876} C_VEL
LIN {X 0,Y 599.866,Z 984.778,A -85,B 0,C 180,E1 978.392,E2 978.392} C_VEL
LIN {X 0,Y 599.858,Z 997.456,A -85,B 0,C 180,E1 981.685,E2 981.685} C_VEL
LIN {X 0,Y 599.798,Z 1005.76,A -85,B 0,C 180,E1 984.95,E2 984.95} C_VEL
LIN {X 0,Y 599.801,Z 1010.09,A -85,B 0,C 180,E1 988.561,E2 988.561} C_VEL
LIN {X 0,Y 599.977,Z 1010.087,A -85,B 0,C 180,E1 991.443,E2 991.443} C_VEL
LIN {X 0,Y 599.992,Z 1005.752,A -85,B 0,C 180,E1 995.053,E2 995.053} C_VEL
LIN {X 0,Y 599.989,Z 995.066,A -85,B 0,C 180,E1 999.047,E2 999.047} C_VEL
LIN {X 0,Y 600.043,Z 979.439,A -85,B 0,C 180,E1 1002.715,E2 1002.715} C_VEL
LIN {X 0,Y 600.116,Z 957.702,A -85,B 0,C 180,E1 1006.336,E2 1006.336} C_VEL
LIN {X 0,Y 600.356,Z 932.052,A -85,B 0,C 180,E1 1009.543,E2 1009.543} C_VEL
LIN {X 0,Y 600.639,Z 901.434,A -85,B 0,C 180,E1 1012.482,E2 1012.482} C_VEL
LIN {X 0,Y 601.007,Z 866.883,A -85,B 0,C 180,E1 1015.002,E2 1015.002} C_VEL
LIN {X 0,Y 601.374,Z 828.834,A -85,B 0,C 180,E1 1017.036,E2 1017.036} C_VEL
LIN {X 0,Y 601.58,Z 789.379,A -85,B 0,C 180,E1 1018.467,E2 1018.467} C_VEL
LIN {X 0,Y 601.823,Z 750.166,A -85,B 0,C 180,E1 1019.274,E2 1019.274} C_VEL
LIN {X 0,Y 601.14,Z 689.289,A -85,B 0,C 180,E1 1020.131,E2 1020.131} C_VEL
LIN {X 0,Y 599.867,Z 685.03,A -85,B 0,C 180,E1 1020.332,E2 1020.332} C_VEL
LIN {X 0,Y 599.397,Z 685.03,A -85,B 0,C 180,E1 1025.387,E2 1025.387} C_VEL
LIN {X 0,Y 599.617,Z 685.03,A -85,B 0,C 180,E1 1028.993,E2 1028.993} C_VEL
LIN {X 0,Y 599.549,Z 685.03,A -85,B 0,C 180,E1 1035.193,E2 1035.193} C_VEL
LIN {X 0,Y 599.556,Z 685.03,A -85,B 0,C 180,E1 1041.008,E2 1041.008} C_VEL
LIN {X 0,Y 599.573,Z 685.03,A -85,B 0,C 180,E1 1044.629,E2 1044.629} C_VEL
LIN {X 0,Y 599.596,Z 685.03,A -85,B 0,C 180,E1 1049.778,E2 1049.778} C_VEL
LIN {X 0,Y 599.863,Z 685.03,A -85,B 0,C 180,E1 1054.917,E2 1054.917} C_VEL
LIN {X 0,Y 599.631,Z 685.03,A -85,B 0,C 180,E1 1060.902,E2 1060.902} C_VEL
LIN {X 0,Y 599.887,Z 685.03,A -85,B 0,C 180,E1 1064.543,E2 1064.543} C_VEL
LIN {X 0,Y 600.493,Z 742.16,A -85,B 0,C 180,E1 1065.396,E2 1065.396} C_VEL
LIN {X 0,Y 600.441,Z 770.47,A -85,B 0,C 180,E1 1066.37,E2 1066.37} C_VEL
LIN {X 0,Y 600.294,Z 796.179,A -85,B 0,C 180,E1 1067.844,E2 1067.844} C_VEL
LIN {X 0,Y 600.198,Z 819.487,A -85,B 0,C 180,E1 1069.861,E2 1069.861} C_VEL
LIN {X 0,Y 600.067,Z 837.923,A -85,B 0,C 180,E1 1072.229,E2 1072.229} C_VEL
LIN {X 0,Y 600.03,Z 849.988,A -85,B 0,C 180,E1 1074.586,E2 1074.586} C_VEL
LIN {X 0,Y 600.045,Z 857.605,A -85,B 0,C 180,E1 1077.114,E2 1077.114} C_VEL
LIN {X 0,Y 599.959,Z 860.489,A -85,B 0,C 180,E1 1079.997,E2 1079.997} C_VEL
LIN {X 0,Y 600.031,Z 857.427,A -85,B 0,C 180,E1 1082.88,E2 1082.88} C_VEL
LIN {X 0,Y 600.037,Z 849.636,A -85,B 0,C 180,E1 1085.408,E2 1085.408} C_VEL
LIN {X 0,Y 600.097,Z 836.192,A -85,B 0,C 180,E1 1087.946,E2 1087.946} C_VEL
LIN {X 0,Y 600.209,Z 817.283,A -85,B 0,C 180,E1 1090.279,E2 1090.279} C_VEL
LIN {X 0,Y 600.314,Z 793.628,A -85,B 0,C 180,E1 1092.241,E2 1092.241} C_VEL
LIN {X 0,Y 600.458,Z 766.452,A -85,B 0,C 180,E1 1093.715,E2 1093.715} C_VEL
LIN {X 0,Y 600.573,Z 737.562,A -85,B 0,C 180,E1 1094.621,E2 1094.621} C_VEL
LIN {X 0,Y 599.935,Z 685.03,A -85,B 0,C 180,E1 1095.402,E2 1095.402} C_VEL
LIN {X 0,Y 599.537,Z 685.03,A -85,B 0,C 180,E1 1101.353,E2 1101.353} C_VEL
LIN {X 0,Y 599.788,Z 685.03,A -85,B 0,C 180,E1 1105.316,E2 1105.316} C_VEL
LIN {X 0,Y 599.5,Z 685.03,A -85,B 0,C 180,E1 1111.141,E2 1111.141} C_VEL
LIN {X 0,Y 599.794,Z 685.03,A -85,B 0,C 180,E1 1117.135,E2 1117.135} C_VEL
LIN {X 0,Y 599.42,Z 685.03,A -85,B 0,C 180,E1 1123.102,E2 1123.102} C_VEL
LIN {X 0,Y 599.58,Z 685.03,A -85,B 0,C 180,E1 1127.188,E2 1127.188} C_VEL
LIN {X 0,Y 599.625,Z 685.03,A -85,B 0,C 180,E1 1132.84,E2 1132.84} C_VEL
LIN {X 0,Y 599.561,Z 685.03,A -85,B 0,C 180,E1 1138.826,E2 1138.826} C_VEL
LIN {X 0,Y 599.864,Z 685.03,A -85,B 0,C 180,E1 1144.887,E2 1144.887} C_VEL
LIN {X 0,Y 599.666,Z 685.183,A -85,B 0,C 180,E1 1149.495,E2 1149.495} C_VEL
LIN {X 0,Y 600.877,Z 710.52,A -85,B 0,C 180,E1 1150.164,E2 1150.164} C_VEL
LIN {X 0,Y 600.663,Z 743.487,A -85,B 0,C 180,E1 1151.505,E2 1151.505} C_VEL
LIN {X 0,Y 600.437,Z 774.383,A -85,B 0,C 180,E1 1153.405,E2 1153.405} C_VEL
LIN {X 0,Y 600.265,Z 800.1,A -85,B 0,C 180,E1 1155.623,E2 1155.623} C_VEL
LIN {X 0,Y 600.123,Z 823.256,A -85,B 0,C 180,E1 1158.392,E2 1158.392} C_VEL
LIN {X 0,Y 599.994,Z 840.456,A -85,B 0,C 180,E1 1161.318,E2 1161.318} C_VEL
LIN {X 0,Y 599.924,Z 851.854,A -85,B 0,C 180,E1 1164.223,E2 1164.223} C_VEL
LIN {X 0,Y 599.888,Z 858.393,A -85,B 0,C 180,E1 1167.114,E2 1167.114} C_VEL
LIN {X 0,Y 599.854,Z 860.497,A -85,B 0,C 180,E1 1169.998,E2 1169.998} C_VEL
LIN {X 0,Y 599.912,Z 858.252,A -85,B 0,C 180,E1 1172.882,E2 1172.882} C_VEL
LIN {X 0,Y 599.952,Z 850.177,A -85,B 0,C 180,E1 1176.22,E2 1176.22} C_VEL
LIN {X 0,Y 599.962,Z 838.239,A -85,B 0,C 180,E1 1179.043,E2 1179.043} C_VEL
LIN {X 0,Y 600.078,Z 819.978,A -85,B 0,C 180,E1 1181.972,E2 1181.972} C_VEL
LIN {X 0,Y 600.256,Z 796.183,A -85,B 0,C 180,E1 1184.67,E2 1184.67} C_VEL
LIN {X 0,Y 600.475,Z 768.89,A -85,B 0,C 180,E1 1186.896,E2 1186.896} C_VEL
LIN {X 0,Y 600.674,Z 737.934,A -85,B 0,C 180,E1 1188.68,E2 1188.68} C_VEL
LIN {X 0,Y 600.879,Z 705.766,A -85,B 0,C 180,E1 1189.886,E2 1189.886} C_VEL
LIN {X 0,Y 599.973,Z 685.03,A -85,B 0,C 180,E1 1190.416,E2 1190.416} C_VEL
LIN {X 0,Y 599.59,Z 685.03,A -85,B 0,C 180,E1 1196.936,E2 1196.936} C_VEL
LIN {X 0,Y 599.721,Z 685.03,A -85,B 0,C 180,E1 1203.611,E2 1203.611} C_VEL
LIN {X 0,Y 599.63,Z 685.03,A -85,B 0,C 180,E1 1208.986,E2 1208.986} C_VEL
LIN {X 0,Y 599.514,Z 685.03,A -85,B 0,C 180,E1 1215.198,E2 1215.198} C_VEL
LIN {X 0,Y 599.515,Z 685.03,A -85,B 0,C 180,E1 1221.013,E2 1221.013} C_VEL
LIN {X 0,Y 599.569,Z 685.03,A -85,B 0,C 180,E1 1224.637,E2 1224.637} C_VEL
LIN {X 0,Y 599.62,Z 685.03,A -85,B 0,C 180,E1 1229.787,E2 1229.787} C_VEL
LIN {X 0,Y 599.831,Z 685.03,A -85,B 0,C 180,E1 1234.913,E2 1234.913} C_VEL
LIN {X 0,Y 599.753,Z 685.03,A -85,B 0,C 180,E1 1240.913,E2 1240.913} C_VEL
LIN {X 0,Y 599.982,Z 685.03,A -85,B 0,C 180,E1 1246.922,E2 1246.922} C_VEL
LIN {X 0,Y 599.709,Z 685.03,A -85,B 0,C 180,E1 1252.776,E2 1252.776} C_VEL
LIN {X 0,Y 599.813,Z 685.03,A -85,B 0,C 180,E1 1257.119,E2 1257.119} C_VEL
LIN {X 0,Y 599.575,Z 685.03,A -85,B 0,C 180,E1 1259.175,E2 1259.175} C_VEL
LIN {X 0,Y 597.199,Z 685.03,A -85,B 0,C 180,E1 1260.411,E2 1260.411} C_VEL
LIN {X 0,Y 591.785,Z 685.03,A -85,B 0,C 180,E1 1262.473,E2 1262.473} C_VEL
LIN {X 0,Y 591.684,Z 685.03,A -85,B 0,C 180,E1 1267.329,E2 1267.329} C_VEL
LIN {X 0,Y 591.685,Z 685.03,A -85,B 0,C 180,E1 1271.775,E2 1271.775} C_VEL
LIN {X 0,Y 591.742,Z 685.03,A -85,B 0,C 180,E1 1276.293,E2 1276.293} C_VEL
LIN {X 0,Y 591.763,Z 685.03,A -85,B 0,C 180,E1 1280.918,E2 1280.918} C_VEL
LIN {X 0,Y 591.52,Z 685.03,A -85,B 0,C 180,E1 1286.763,E2 1286.763} C_VEL
LIN {X 0,Y 591.652,Z 685.03,A -85,B 0,C 180,E1 1290.671,E2 1290.671} C_VEL
LIN {X 0,Y 591.713,Z 685.03,A -85,B 0,C 180,E1 1295.913,E2 1295.913} C_VEL
LIN {X 0,Y 591.64,Z 685.03,A -85,B 0,C 180,E1 1301.54,E2 1301.54} C_VEL
LIN {X 0,Y 591.505,Z 685.03,A -85,B 0,C 180,E1 1306.465,E2 1306.465} C_VEL
LIN {X 0,Y 591.525,Z 685.03,A -85,B 0,C 180,E1 1312.261,E2 1312.261} C_VEL
LIN {X 0,Y 591.792,Z 685.03,A -85,B 0,C 180,E1 1317.625,E2 1317.625} C_VEL
LIN {X 0,Y 591.919,Z 685.635,A -85,B 0,C 180,E1 1319.299,E2 1319.299} C_VEL
LIN {X 0,Y 594.681,Z 695.02,A -85,B 0,C 180,E1 1319.586,E2 1319.586} C_VEL
LIN {X 0,Y 594.673,Z 773.379,A -85,B 0,C 180,E1 1320.762,E2 1320.762} C_VEL
LIN {X 0,Y 594.432,Z 810.346,A -85,B 0,C 180,E1 1321.86,E2 1321.86} C_VEL
LIN {X 0,Y 594.008,Z 844.97,A -85,B 0,C 180,E1 1323.402,E2 1323.402} C_VEL
LIN {X 0,Y 593.459,Z 879.795,A -85,B 0,C 180,E1 1325.537,E2 1325.537} C_VEL
LIN {X 0,Y 592.955,Z 913.088,A -85,B 0,C 180,E1 1328.258,E2 1328.258} C_VEL
LIN {X 0,Y 592.52,Z 941.14,A -85,B 0,C 180,E1 1331.246,E2 1331.246} C_VEL
LIN {X 0,Y 592.161,Z 964.559,A -85,B 0,C 180,E1 1334.482,E2 1334.482} C_VEL
LIN {X 0,Y 591.991,Z 983.036,A -85,B 0,C 180,E1 1337.862,E2 1337.862} C_VEL
LIN {X 0,Y 591.993,Z 996.313,A -85,B 0,C 180,E1 1341.204,E2 1341.204} C_VEL
LIN {X 0,Y 591.921,Z 1005.759,A -85,B 0,C 180,E1 1344.883,E2 1344.883} C_VEL
LIN {X 0,Y 591.9,Z 1010.092,A -85,B 0,C 180,E1 1348.541,E2 1348.541} C_VEL
LIN {X 0,Y 592.071,Z 1010.089,A -85,B 0,C 180,E1 1351.463,E2 1351.463} C_VEL
LIN {X 0,Y 592.091,Z 1005.751,A -85,B 0,C 180,E1 1355.12,E2 1355.12} C_VEL
LIN {X 0,Y 592.104,Z 995.068,A -85,B 0,C 180,E1 1359.168,E2 1359.168} C_VEL
LIN {X 0,Y 592.19,Z 979.441,A -85,B 0,C 180,E1 1362.886,E2 1362.886} C_VEL
LIN {X 0,Y 592.352,Z 957.937,A -85,B 0,C 180,E1 1366.523,E2 1366.523} C_VEL
LIN {X 0,Y 592.674,Z 931.97,A -85,B 0,C 180,E1 1369.817,E2 1369.817} C_VEL
LIN {X 0,Y 593.12,Z 901.731,A -85,B 0,C 180,E1 1372.757,E2 1372.757} C_VEL
LIN {X 0,Y 593.679,Z 867.689,A -85,B 0,C 180,E1 1375.279,E2 1375.279} C_VEL
LIN {X 0,Y 594.19,Z 831.305,A -85,B 0,C 180,E1 1377.272,E2 1377.272} C_VEL
LIN {X 0,Y 594.574,Z 794.032,A -85,B 0,C 180,E1 1378.69,E2 1378.69} C_VEL
LIN {X 0,Y 594.902,Z 756.822,A -85,B 0,C 180,E1 1379.543,E2 1379.543} C_VEL
LIN {X 0,Y 594.177,Z 691.583,A -85,B 0,C 180,E1 1380.49,E2 1380.49} C_VEL
LIN {X 0,Y 591.936,Z 685.03,A -85,B 0,C 180,E1 1380.775,E2 1380.775} C_VEL
LIN {X 0,Y 591.433,Z 685.03,A -85,B 0,C 180,E1 1385.937,E2 1385.937} C_VEL
LIN {X 0,Y 591.462,Z 685.03,A -85,B 0,C 180,E1 1391.561,E2 1391.561} C_VEL
LIN {X 0,Y 591.634,Z 685.03,A -85,B 0,C 180,E1 1396.477,E2 1396.477} C_VEL
LIN {X 0,Y 591.687,Z 685.03,A -85,B 0,C 180,E1 1402.26,E2 1402.26} C_VEL
LIN {X 0,Y 591.451,Z 685.03,A -85,B 0,C 180,E1 1407.602,E2 1407.602} C_VEL
LIN {X 0,Y 591.526,Z 685.03,A -85,B 0,C 180,E1 1412.664,E2 1412.664} C_VEL
LIN {X 0,Y 591.506,Z 685.03,A -85,B 0,C 180,E1 1417.5,E2 1417.5} C_VEL
LIN {X 0,Y 591.552,Z 685.03,A -85,B 0,C 180,E1 1422.173,E2 1422.173} C_VEL
LIN {X 0,Y 591.929,Z 685.03,A -85,B 0,C 180,E1 1424.33,E2 1424.33} C_VEL
LIN {X 0,Y 592.911,Z 713.223,A -85,B 0,C 180,E1 1424.735,E2 1424.735} C_VEL
LIN {X 0,Y 592.825,Z 746.715,A -85,B 0,C 180,E1 1425.32,E2 1425.32} C_VEL
LIN {X 0,Y 592.676,Z 774.656,A -85,B 0,C 180,E1 1426.393,E2 1426.393} C_VEL
LIN {X 0,Y 592.492,Z 801.189,A -85,B 0,C 180,E1 1428.055,E2 1428.055} C_VEL
LIN {X 0,Y 592.297,Z 822.815,A -85,B 0,C 180,E1 1430.095,E2 1430.095} C_VEL
LIN {X 0,Y 592.146,Z 840.122,A -85,B 0,C 180,E1 1432.493,E2 1432.493} C_VEL
LIN {X 0,Y 592.096,Z 851.383,A -85,B 0,C 180,E1 1434.88,E2 1434.88} C_VEL
LIN {X 0,Y 592.144,Z 857.607,A -85,B 0,C 180,E1 1437.076,E2 1437.076} C_VEL
LIN {X 0,Y 592.059,Z 860.481,A -85,B 0,C 180,E1 1439.997,E2 1439.997} C_VEL
LIN {X 0,Y 592.129,Z 857.431,A -85,B 0,C 180,E1 1442.918,E2 1442.918} C_VEL
LIN {X 0,Y 592.154,Z 849.635,A -85,B 0,C 180,E1 1445.48,E2 1445.48} C_VEL
LIN {X 0,Y 592.25,Z 836.197,A -85,B 0,C 180,E1 1448.052,E2 1448.052} C_VEL
LIN {X 0,Y 592.396,Z 817.509,A -85,B 0,C 180,E1 1450.393,E2 1450.393} C_VEL
LIN {X 0,Y 592.546,Z 793.642,A -85,B 0,C 180,E1 1452.404,E2 1452.404} C_VEL
LIN {X 0,Y 592.752,Z 766.898,A -85,B 0,C 180,E1 1453.878,E2 1453.878} C_VEL
LIN {X 0,Y 592.934,Z 737.51,A -85,B 0,C 180,E1 1454.815,E2 1454.815} C_VEL
LIN {X 0,Y 591.955,Z 685.03,A -85,B 0,C 180,E1 1455.561,E2 1455.561} C_VEL
LIN {X 0,Y 591.775,Z 685.03,A -85,B 0,C 180,E1 1460.91,E2 1460.91} C_VEL
LIN {X 0,Y 591.539,Z 685.03,A -85,B 0,C 180,E1 1466.757,E2 1466.757} C_VEL
LIN {X 0,Y 591.629,Z 685.03,A -85,B 0,C 180,E1 1470.665,E2 1470.665} C_VEL
LIN {X 0,Y 591.756,Z 685.03,A -85,B 0,C 180,E1 1475.902,E2 1475.902} C_VEL
LIN {X 0,Y 591.582,Z 685.03,A -85,B 0,C 180,E1 1480.065,E2 1480.065} C_VEL
LIN {X 0,Y 591.61,Z 685.03,A -85,B 0,C 180,E1 1485.567,E2 1485.567} C_VEL
LIN {X 0,Y 591.556,Z 685.03,A -85,B 0,C 180,E1 1490.372,E2 1490.372} C_VEL
LIN {X 0,Y 591.462,Z 685.03,A -85,B 0,C 180,E1 1495.85,E2 1495.85} C_VEL
LIN {X 0,Y 591.579,Z 685.03,A -85,B 0,C 180,E1 1501.006,E2 1501.006} C_VEL
LIN {X 0,Y 591.698,Z 685.03,A -85,B 0,C 180,E1 1505.914,E2 1505.914} C_VEL
LIN {X 0,Y 591.705,Z 685.03,A -85,B 0,C 180,E1 1509.197,E2 1509.197} C_VEL
LIN {X 0,Y 593.487,Z 700.596,A -85,B 0,C 180,E1 1509.619,E2 1509.619} C_VEL
LIN {X 0,Y 593.174,Z 734.569,A -85,B 0,C 180,E1 1510.829,E2 1510.829} C_VEL
LIN {X 0,Y 592.858,Z 765.624,A -85,B 0,C 180,E1 1512.562,E2 1512.562} C_VEL
LIN {X 0,Y 592.564,Z 793.366,A -85,B 0,C 180,E1 1514.772,E2 1514.772} C_VEL
LIN {X 0,Y 592.26,Z 816.388,A -85,B 0,C 180,E1 1517.302,E2 1517.302} C_VEL
LIN {X 0,Y 592.134,Z 834.793,A -85,B 0,C 180,E1 1520.092,E2 1520.092} C_VEL
LIN {X 0,Y 592.009,Z 849.123,A -85,B 0,C 180,E1 1523.303,E2 1523.303} C_VEL
LIN {X 0,Y 592.04,Z 857.205,A -85,B 0,C 180,E1 1526.344,E2 1526.344} C_VEL
LIN {X 0,Y 592.047,Z 859.949,A -85,B 0,C 180,E1 1528.537,E2 1528.537} C_VEL
LIN {X 0,Y 592.051,Z 859.89,A -85,B 0,C 180,E1 1531.458,E2 1531.458} C_VEL
LIN {X 0,Y 592.056,Z 855.511,A -85,B 0,C 180,E1 1534.383,E2 1534.383} C_VEL
LIN {X 0,Y 592.16,Z 844.992,A -85,B 0,C 180,E1 1537.687,E2 1537.687} C_VEL
LIN {X 0,Y 592.267,Z 828.972,A -85,B 0,C 180,E1 1540.805,E2 1540.805} C_VEL
LIN {X 0,Y 592.463,Z 808.286,A -85,B 0,C 180,E1 1543.59,E2 1543.59} C_VEL
LIN {X 0,Y 592.68,Z 782.701,A -85,B 0,C 180,E1 1546.073,E2 1546.073} C_VEL
LIN {X 0,Y 592.984,Z 752.485,A -85,B 0,C 180,E1 1548.162,E2 1548.162} C_VEL
LIN {X 0,Y 593.268,Z 719.624,A -85,B 0,C 180,E1 1549.697,E2 1549.697} C_VEL
LIN {X 0,Y 592.906,Z 688.705,A -85,B 0,C 180,E1 1550.59,E2 1550.59} C_VEL
LIN {X 0,Y 592.021,Z 685.03,A -85,B 0,C 180,E1 1550.746,E2 1550.746} C_VEL
LIN {X 0,Y 591.708,Z 685.03,A -85,B 0,C 180,E1 1557.324,E2 1557.324} C_VEL
LIN {X 0,Y 591.714,Z 685.03,A -85,B 0,C 180,E1 1564.128,E2 1564.128} C_VEL
LIN {X 0,Y 591.527,Z 685.03,A -85,B 0,C 180,E1 1570.077,E2 1570.077} C_VEL
LIN {X 0,Y 591.577,Z 685.03,A -85,B 0,C 180,E1 1575.58,E2 1575.58} C_VEL
LIN {X 0,Y 591.562,Z 685.03,A -85,B 0,C 180,E1 1580.386,E2 1580.386} C_VEL
LIN {X 0,Y 591.497,Z 685.03,A -85,B 0,C 180,E1 1585.865,E2 1585.865} C_VEL
LIN {X 0,Y 591.56,Z 685.03,A -85,B 0,C 180,E1 1591.016,E2 1591.016} C_VEL
LIN {X 0,Y 591.634,Z 685.03,A -85,B 0,C 180,E1 1595.921,E2 1595.921} C_VEL
LIN {X 0,Y 591.829,Z 685.03,A -85,B 0,C 180,E1 1600.648,E2 1600.648} C_VEL
LIN {X 0,Y 592.036,Z 685.03,A -85,B 0,C 180,E1 1606.743,E2 1606.743} C_VEL
LIN {X 0,Y 591.814,Z 685.03,A -85,B 0,C 180,E1 1612.731,E2 1612.731} C_VEL
LIN {X 0,Y 591.906,Z 685.03,A -85,B 0,C 180,E1 1617.081,E2 1617.081} C_VEL
LIN {X 0,Y 591.785,Z 685.03,A -85,B 0,C 180,E1 1622.473,E2 1622.473} C_VEL
LIN {X 0,Y 587.737,Z 685.03,A -85,B 0,C 180,E1 1624.13,E2 1624.13} C_VEL
LIN {X 0,Y 584.087,Z 685.03,A -85,B 0,C 180,E1 1625.809,E2 1625.809} C_VEL
LIN {X 0,Y 583.777,Z 685.03,A -85,B 0,C 180,E1 1631.937,E2 1631.937} C_VEL
LIN {X 0,Y 583.724,Z 685.03,A -85,B 0,C 180,E1 1636.96,E2 1636.96} C_VEL
LIN {X 0,Y 583.724,Z 685.03,A -85,B 0,C 180,E1 1641.463,E2 1641.463} C_VEL
LIN {X 0,Y 583.726,Z 685.03,A -85,B 0,C 180,E1 1646.071,E2 1646.071} C_VEL
LIN {X 0,Y 583.594,Z 685.03,A -85,B 0,C 180,E1 1651.429,E2 1651.429} C_VEL
LIN {X 0,Y 583.748,Z 685.03,A -85,B 0,C 180,E1 1656.74,E2 1656.74} C_VEL
LIN {X 0,Y 583.738,Z 685.03,A -85,B 0,C 180,E1 1662.231,E2 1662.231} C_VEL
LIN {X 0,Y 583.543,Z 685.03,A -85,B 0,C 180,E1 1667.752,E2 1667.752} C_VEL
LIN {X 0,Y 583.51,Z 685.03,A -85,B 0,C 180,E1 1673.29,E2 1673.29} C_VEL
LIN {X 0,Y 583.973,Z 685.03,A -85,B 0,C 180,E1 1678.775,E2 1678.775} C_VEL
LIN {X 0,Y 587.862,Z 696.417,A -85,B 0,C 180,E1 1679.214,E2 1679.214} C_VEL
LIN {X 0,Y 587.774,Z 773.504,A -85,B 0,C 180,E1 1680.387,E2 1680.387} C_VEL
LIN {X 0,Y 587.38,Z 810.758,A -85,B 0,C 180,E1 1681.506,E2 1681.506} C_VEL
LIN {X 0,Y 586.771,Z 847.187,A -85,B 0,C 180,E1 1683.17,E2 1683.17} C_VEL
LIN {X 0,Y 586.023,Z 882.44,A -85,B 0,C 180,E1 1685.402,E2 1685.402} C_VEL
LIN {X 0,Y 585.359,Z 914.845,A -85,B 0,C 180,E1 1688.129,E2 1688.129} C_VEL
LIN {X 0,Y 584.788,Z 944.31,A -85,B 0,C 180,E1 1691.379,E2 1691.379} C_VEL
LIN {X 0,Y 584.39,Z 968.093,A -85,B 0,C 180,E1 1694.846,E2 1694.846} C_VEL
LIN {X 0,Y 584.145,Z 987.059,A -85,B 0,C 180,E1 1698.6,E2 1698.6} C_VEL
LIN {X 0,Y 584.101,Z 999.721,A -85,B 0,C 180,E1 1702.207,E2 1702.207} C_VEL
LIN {X 0,Y 583.998,Z 1006.968,A -85,B 0,C 180,E1 1705.556,E2 1705.556} C_VEL
LIN {X 0,Y 584.025,Z 1010.094,A -85,B 0,C 180,E1 1708.522,E2 1708.522} C_VEL
LIN {X 0,Y 584.181,Z 1010.091,A -85,B 0,C 180,E1 1711.483,E2 1711.483} C_VEL
LIN {X 0,Y 584.209,Z 1005.75,A -85,B 0,C 180,E1 1715.189,E2 1715.189} C_VEL
LIN {X 0,Y 584.198,Z 995.071,A -85,B 0,C 180,E1 1719.293,E2 1719.293} C_VEL
LIN {X 0,Y 584.33,Z 979.444,A -85,B 0,C 180,E1 1723.063,E2 1723.063} C_VEL
LIN {X 0,Y 584.558,Z 958.386,A -85,B 0,C 180,E1 1726.686,E2 1726.686} C_VEL
LIN {X 0,Y 585.024,Z 932.76,A -85,B 0,C 180,E1 1729.999,E2 1729.999} C_VEL
LIN {X 0,Y 585.615,Z 902.253,A -85,B 0,C 180,E1 1733.02,E2 1733.02} C_VEL
LIN {X 0,Y 586.328,Z 868.674,A -85,B 0,C 180,E1 1735.553,E2 1735.553} C_VEL
LIN {X 0,Y 587.029,Z 832.685,A -85,B 0,C 180,E1 1737.566,E2 1737.566} C_VEL
LIN {X 0,Y 587.585,Z 795.352,A -85,B 0,C 180,E1 1739.021,E2 1739.021} C_VEL
LIN {X 0,Y 588.046,Z 758.805,A -85,B 0,C 180,E1 1739.89,E2 1739.89} C_VEL
LIN {X 0,Y 587.393,Z 693.838,A -85,B 0,C 180,E1 1740.849,E2 1740.849} C_VEL
LIN {X 0,Y 584.014,Z 685.03,A -85,B 0,C 180,E1 1741.178,E2 1741.178} C_VEL
LIN {X 0,Y 583.497,Z 685.03,A -85,B 0,C 180,E1 1746.708,E2 1746.708} C_VEL
LIN {X 0,Y 583.565,Z 685.03,A -85,B 0,C 180,E1 1752.252,E2 1752.252} C_VEL
LIN {X 0,Y 583.741,Z 685.03,A -85,B 0,C 180,E1 1757.77,E2 1757.77} C_VEL
LIN {X 0,Y 583.754,Z 685.03,A -85,B 0,C 180,E1 1763.519,E2 1763.519} C_VEL
LIN {X 0,Y 583.638,Z 685.03,A -85,B 0,C 180,E1 1768.861,E2 1768.861} C_VEL
LIN {X 0,Y 583.797,Z 685.03,A -85,B 0,C 180,E1 1774.792,E2 1774.792} C_VEL
LIN {X 0,Y 583.828,Z 685.03,A -85,B 0,C 180,E1 1780.365,E2 1780.365} C_VEL
LIN {X 0,Y 583.955,Z 685.03,A -85,B 0,C 180,E1 1784.134,E2 1784.134} C_VEL
LIN {X 0,Y 585.276,Z 701.649,A -85,B 0,C 180,E1 1784.387,E2 1784.387} C_VEL
LIN {X 0,Y 585.189,Z 744.053,A -85,B 0,C 180,E1 1785.054,E2 1785.054} C_VEL
LIN {X 0,Y 585.022,Z 772.594,A -85,B 0,C 180,E1 1786.108,E2 1786.108} C_VEL
LIN {X 0,Y 584.726,Z 798.689,A -85,B 0,C 180,E1 1787.705,E2 1787.705} C_VEL
LIN {X 0,Y 584.517,Z 821.197,A -85,B 0,C 180,E1 1789.774,E2 1789.774} C_VEL
LIN {X 0,Y 584.316,Z 839.035,A -85,B 0,C 180,E1 1792.205,E2 1792.205} C_VEL
LIN {X 0,Y 584.238,Z 851.383,A -85,B 0,C 180,E1 1794.811,E2 1794.811} C_VEL
LIN {X 0,Y 584.257,Z 857.609,A -85,B 0,C 180,E1 1797.036,E2 1797.036} C_VEL
LIN {X 0,Y 584.17,Z 860.472,A -85,B 0,C 180,E1 1799.997,E2 1799.997} C_VEL
LIN {X 0,Y 584.242,Z 857.435,A -85,B 0,C 180,E1 1802.957,E2 1802.957} C_VEL
LIN {X 0,Y 584.272,Z 849.635,A -85,B 0,C 180,E1 1805.554,E2 1805.554} C_VEL
LIN {X 0,Y 584.378,Z 836.202,A -85,B 0,C 180,E1 1808.161,E2 1808.161} C_VEL
LIN {X 0,Y 584.577,Z 818.71,A -85,B 0,C 180,E1 1810.406,E2 1810.406} C_VEL
LIN {X 0,Y 584.798,Z 796.286,A -85,B 0,C 180,E1 1812.381,E2 1812.381} C_VEL
LIN {X 0,Y 585.025,Z 770.705,A -85,B 0,C 180,E1 1813.895,E2 1813.895} C_VEL
LIN {X 0,Y 585.23,Z 742.476,A -85,B 0,C 180,E1 1814.893,E2 1814.893} C_VEL
LIN {X 0,Y 584.724,Z 688.532,A -85,B 0,C 180,E1 1815.702,E2 1815.702} C_VEL
LIN {X 0,Y 583.994,Z 685.03,A -85,B 0,C 180,E1 1815.834,E2 1815.834} C_VEL
LIN {X 0,Y 583.739,Z 685.03,A -85,B 0,C 180,E1 1821.454,E2 1821.454} C_VEL
LIN {X 0,Y 583.776,Z 685.03,A -85,B 0,C 180,E1 1826.062,E2 1826.062} C_VEL
LIN {X 0,Y 583.574,Z 685.03,A -85,B 0,C 180,E1 1831.417,E2 1831.417} C_VEL
LIN {X 0,Y 583.846,Z 685.03,A -85,B 0,C 180,E1 1836.745,E2 1836.745} C_VEL
LIN {X 0,Y 583.556,Z 685.03,A -85,B 0,C 180,E1 1842.238,E2 1842.238} C_VEL
LIN {X 0,Y 583.726,Z 685.03,A -85,B 0,C 180,E1 1847.762,E2 1847.762} C_VEL
LIN {X 0,Y 583.708,Z 685.03,A -85,B 0,C 180,E1 1853.511,E2 1853.511} C_VEL
LIN {X 0,Y 583.666,Z 685.03,A -85,B 0,C 180,E1 1858.859,E2 1858.859} C_VEL
LIN {X 0,Y 583.836,Z 685.03,A -85,B 0,C 180,E1 1864.754,E2 1864.754} C_VEL
LIN {X 0,Y 583.783,Z 685.422,A -85,B 0,C 180,E1 1868.916,E2 1868.916} C_VEL
LIN {X 0,Y 586.012,Z 698.843,A -85,B 0,C 180,E1 1869.302,E2 1869.302} C_VEL
LIN {X 0,Y 585.686,Z 732.449,A -85,B 0,C 180,E1 1870.477,E2 1870.477} C_VEL
LIN {X 0,Y 585.278,Z 763.439,A -85,B 0,C 180,E1 1872.181,E2 1872.181} C_VEL
LIN {X 0,Y 584.854,Z 791.293,A -85,B 0,C 180,E1 1874.374,E2 1874.374} C_VEL
LIN {X 0,Y 584.499,Z 814.925,A -85,B 0,C 180,E1 1876.941,E2 1876.941} C_VEL
LIN {X 0,Y 584.297,Z 833.738,A -85,B 0,C 180,E1 1879.77,E2 1879.77} C_VEL
LIN {X 0,Y 584.212,Z 846.847,A -85,B 0,C 180,E1 1882.577,E2 1882.577} C_VEL
LIN {X 0,Y 584.197,Z 855.69,A -85,B 0,C 180,E1 1885.553,E2 1885.553} C_VEL
LIN {X 0,Y 584.158,Z 859.949,A -85,B 0,C 180,E1 1888.517,E2 1888.517} C_VEL
LIN {X 0,Y 584.162,Z 859.891,A -85,B 0,C 180,E1 1891.478,E2 1891.478} C_VEL
LIN {X 0,Y 584.159,Z 855.513,A -85,B 0,C 180,E1 1894.443,E2 1894.443} C_VEL
LIN {X 0,Y 584.288,Z 844.996,A -85,B 0,C 180,E1 1897.791,E2 1897.791} C_VEL
LIN {X 0,Y 584.422,Z 828.541,A -85,B 0,C 180,E1 1901.021,E2 1901.021} C_VEL
LIN {X 0,Y 584.709,Z 807.343,A -85,B 0,C 180,E1 1903.886,E2 1903.886} C_VEL
LIN {X 0,Y 585.028,Z 781.574,A -85,B 0,C 180,E1 1906.385,E2 1906.385} C_VEL
LIN {X 0,Y 585.419,Z 752.501,A -85,B 0,C 180,E1 1908.405,E2 1908.405} C_VEL
LIN {X 0,Y 585.801,Z 719.633,A -85,B 0,C 180,E1 1909.959,E2 1909.959} C_VEL
LIN {X 0,Y 585.232,Z 689.814,A -85,B 0,C 180,E1 1910.851,E2 1910.851} C_VEL
LIN {X 0,Y 584.081,Z 685.03,A -85,B 0,C 180,E1 1911.068,E2 1911.068} C_VEL
LIN {X 0,Y 583.743,Z 685.03,A -85,B 0,C 180,E1 1917.729,E2 1917.729} C_VEL
LIN {X 0,Y 583.808,Z 685.03,A -85,B 0,C 180,E1 1924.209,E2 1924.209} C_VEL
LIN {X 0,Y 583.594,Z 685.03,A -85,B 0,C 180,E1 1930.272,E2 1930.272} C_VEL
LIN {X 0,Y 583.704,Z 685.03,A -85,B 0,C 180,E1 1936.374,E2 1936.374} C_VEL
LIN {X 0,Y 583.691,Z 685.03,A -85,B 0,C 180,E1 1941.658,E2 1941.658} C_VEL
LIN {X 0,Y 583.57,Z 685.03,A -85,B 0,C 180,E1 1947.118,E2 1947.118} C_VEL
LIN {X 0,Y 583.622,Z 685.03,A -85,B 0,C 180,E1 1952.27,E2 1952.27} C_VEL
LIN {X 0,Y 583.6,Z 685.03,A -85,B 0,C 180,E1 1957.185,E2 1957.185} C_VEL
LIN {X 0,Y 583.86,Z 685.03,A -85,B 0,C 180,E1 1961.937,E2 1961.937} C_VEL
LIN {X 0,Y 584.116,Z 685.03,A -85,B 0,C 180,E1 1966.56,E2 1966.56} C_VEL
LIN {X 0,Y 583.891,Z 685.03,A -85,B 0,C 180,E1 1972.715,E2 1972.715} C_VEL
LIN {X 0,Y 584.024,Z 685.03,A -85,B 0,C 180,E1 1977.041,E2 1977.041} C_VEL
LIN {X 0,Y 583.902,Z 685.03,A -85,B 0,C 180,E1 1982.459,E2 1982.459} C_VEL
LIN {X 0,Y 584.087,Z 685.03,A -85,B 0,C 180,E1 1985.809,E2 1985.809} C_VEL
LIN {X 0,Y 581.625,Z 685.03,A -85,B 0,C 180,E1 1987.069,E2 1987.069} C_VEL
LIN {X 0,Y 575.965,Z 685.03,A -85,B 0,C 180,E1 1988.954,E2 1988.954} C_VEL
LIN {X 0,Y 575.862,Z 685.03,A -85,B 0,C 180,E1 1989.172,E2 1989.172} C_VEL
LIN {X 0,Y 575.937,Z 685.03,A -85,B 0,C 180,E1 1995.191,E2 1995.191} C_VEL
LIN {X 0,Y 575.83,Z 685.03,A -85,B 0,C 180,E1 2001.525,E2 2001.525} C_VEL
LIN {X 0,Y 575.668,Z 685.03,A -85,B 0,C 180,E1 2006.969,E2 2006.969} C_VEL
LIN {X 0,Y 575.685,Z 685.03,A -85,B 0,C 180,E1 2011.618,E2 2011.618} C_VEL
LIN {X 0,Y 575.83,Z 685.03,A -85,B 0,C 180,E1 2017.066,E2 2017.066} C_VEL
LIN {X 0,Y 575.801,Z 685.03,A -85,B 0,C 180,E1 2022.952,E2 2022.952} C_VEL
LIN {X 0,Y 575.651,Z 685.03,A -85,B 0,C 180,E1 2029.055,E2 2029.055} C_VEL
LIN {X 0,Y 575.703,Z 685.03,A -85,B 0,C 180,E1 2034.785,E2 2034.785} C_VEL
LIN {X 0,Y 576.025,Z 685.121,A -85,B 0,C 180,E1 2038.348,E2 2038.348} C_VEL
LIN {X 0,Y 581.079,Z 699.376,A -85,B 0,C 180,E1 2038.857,E2 2038.857} C_VEL
LIN {X 0,Y 580.911,Z 773.529,A -85,B 0,C 180,E1 2040.002,E2 2040.002} C_VEL
LIN {X 0,Y 580.344,Z 812.144,A -85,B 0,C 180,E1 2041.181,E2 2041.181} C_VEL
LIN {X 0,Y 579.548,Z 849.234,A -85,B 0,C 180,E1 2042.922,E2 2042.922} C_VEL
LIN {X 0,Y 578.599,Z 885.046,A -85,B 0,C 180,E1 2045.26,E2 2045.26} C_VEL
LIN {X 0,Y 577.754,Z 917.917,A -85,B 0,C 180,E1 2048.128,E2 2048.128} C_VEL
LIN {X 0,Y 577.065,Z 945.971,A -85,B 0,C 180,E1 2051.341,E2 2051.341} C_VEL
LIN {X 0,Y 576.557,Z 969.189,A -85,B 0,C 180,E1 2054.829,E2 2054.829} C_VEL
LIN {X 0,Y 576.273,Z 986.784,A -85,B 0,C 180,E1 2058.373,E2 2058.373} C_VEL
LIN {X 0,Y 576.205,Z 999.72,A -85,B 0,C 180,E1 2062.099,E2 2062.099} C_VEL
LIN {X 0,Y 576.099,Z 1006.97,A -85,B 0,C 180,E1 2065.495,E2 2065.495} C_VEL
LIN {X 0,Y 576.124,Z 1010.096,A -85,B 0,C 180,E1 2068.501,E2 2068.501} C_VEL
LIN {X 0,Y 576.275,Z 1010.093,A -85,B 0,C 180,E1 2071.503,E2 2071.503} C_VEL
LIN {X 0,Y 576.253,Z 1004.875,A -85,B 0,C 180,E1 2075.699,E2 2075.699} C_VEL
LIN {X 0,Y 576.29,Z 995.073,A -85,B 0,C 180,E1 2079.422,E2 2079.422} C_VEL
LIN {X 0,Y 576.467,Z 979.446,A -85,B 0,C 180,E1 2083.244,E2 2083.244} C_VEL
LIN {X 0,Y 576.774,Z 958.389,A -85,B 0,C 180,E1 2086.918,E2 2086.918} C_VEL
LIN {X 0,Y 577.386,Z 932.858,A -85,B 0,C 180,E1 2090.264,E2 2090.264} C_VEL
LIN {X 0,Y 578.127,Z 902.615,A -85,B 0,C 180,E1 2093.304,E2 2093.304} C_VEL
LIN {X 0,Y 579.032,Z 868.68,A -85,B 0,C 180,E1 2095.898,E2 2095.898} C_VEL
LIN {X 0,Y 579.911,Z 832.691,A -85,B 0,C 180,E1 2097.934,E2 2097.934} C_VEL
LIN {X 0,Y 580.623,Z 795.358,A -85,B 0,C 180,E1 2099.403,E2 2099.403} C_VEL
LIN {X 0,Y 581.194,Z 760.567,A -85,B 0,C 180,E1 2100.25,E2 2100.25} C_VEL
LIN {X 0,Y 580.586,Z 696.397,A -85,B 0,C 180,E1 2101.215,E2 2101.215} C_VEL
LIN {X 0,Y 576.068,Z 685.03,A -85,B 0,C 180,E1 2101.693,E2 2101.693} C_VEL
LIN {X 0,Y 575.638,Z 685.03,A -85,B 0,C 180,E1 2108.148,E2 2108.148} C_VEL
LIN {X 0,Y 575.682,Z 685.03,A -85,B 0,C 180,E1 2112.969,E2 2112.969} C_VEL
LIN {X 0,Y 575.785,Z 685.03,A -85,B 0,C 180,E1 2119.066,E2 2119.066} C_VEL
LIN {X 0,Y 575.712,Z 685.03,A -85,B 0,C 180,E1 2124.785,E2 2124.785} C_VEL
LIN {X 0,Y 575.715,Z 685.03,A -85,B 0,C 180,E1 2130.131,E2 2130.131} C_VEL
LIN {X 0,Y 575.863,Z 685.03,A -85,B 0,C 180,E1 2135.21,E2 2135.21} C_VEL
LIN {X 0,Y 575.871,Z 685.03,A -85,B 0,C 180,E1 2140.635,E2 2140.635} C_VEL
LIN {X 0,Y 575.987,Z 685.03,A -85,B 0,C 180,E1 2143.909,E2 2143.909} C_VEL
LIN {X 0,Y 577.685,Z 697.758,A -85,B 0,C 180,E1 2144.128,E2 2144.128} C_VEL
LIN {X 0,Y 577.581,Z 742.066,A -85,B 0,C 180,E1 2144.804,E2 2144.804} C_VEL
LIN {X 0,Y 577.342,Z 770.401,A -85,B 0,C 180,E1 2145.812,E2 2145.812} C_VEL
LIN {X 0,Y 576.987,Z 796.106,A -85,B 0,C 180,E1 2147.345,E2 2147.345} C_VEL
LIN {X 0,Y 576.75,Z 819.482,A -85,B 0,C 180,E1 2149.444,E2 2149.444} C_VEL
LIN {X 0,Y 576.487,Z 837.881,A -85,B 0,C 180,E1 2151.909,E2 2151.909} C_VEL
LIN {X 0,Y 576.382,Z 850.539,A -85,B 0,C 180,E1 2154.504,E2 2154.504} C_VEL
LIN {X 0,Y 576.356,Z 857.61,A -85,B 0,C 180,E1 2156.995,E2 2156.995} C_VEL
LIN {X 0,Y 576.27,Z 860.464,A -85,B 0,C 180,E1 2159.997,E2 2159.997} C_VEL
LIN {X 0,Y 576.341,Z 857.44,A -85,B 0,C 180,E1 2162.998,E2 2162.998} C_VEL
LIN {X 0,Y 576.368,Z 849.17,A -85,B 0,C 180,E1 2165.745,E2 2165.745} C_VEL
LIN {X 0,Y 576.496,Z 835.004,A -85,B 0,C 180,E1 2168.463,E2 2168.463} C_VEL
LIN {X 0,Y 576.765,Z 815.689,A -85,B 0,C 180,E1 2170.863,E2 2170.863} C_VEL
LIN {X 0,Y 577.067,Z 792.298,A -85,B 0,C 180,E1 2172.838,E2 2172.838} C_VEL
LIN {X 0,Y 577.373,Z 766.09,A -85,B 0,C 180,E1 2174.29,E2 2174.29} C_VEL
LIN {X 0,Y 577.67,Z 736.688,A -85,B 0,C 180,E1 2175.235,E2 2175.235} C_VEL
LIN {X 0,Y 576.867,Z 688.908,A -85,B 0,C 180,E1 2175.918,E2 2175.918} C_VEL
LIN {X 0,Y 576.003,Z 685.03,A -85,B 0,C 180,E1 2176.059,E2 2176.059} C_VEL
LIN {X 0,Y 575.846,Z 685.03,A -85,B 0,C 180,E1 2181.517,E2 2181.517} C_VEL
LIN {X 0,Y 575.691,Z 685.03,A -85,B 0,C 180,E1 2186.964,E2 2186.964} C_VEL
LIN {X 0,Y 575.665,Z 685.03,A -85,B 0,C 180,E1 2191.612,E2 2191.612} C_VEL
LIN {X 0,Y 575.935,Z 685.03,A -85,B 0,C 180,E1 2197.05,E2 2197.05} C_VEL
LIN {X 0,Y 575.666,Z 685.03,A -85,B 0,C 180,E1 2202.955,E2 2202.955} C_VEL
LIN {X 0,Y 575.787,Z 685.03,A -85,B 0,C 180,E1 2209.06,E2 2209.06} C_VEL
LIN {X 0,Y 575.672,Z 685.03,A -85,B 0,C 180,E1 2214.778,E2 2214.778} C_VEL
LIN {X 0,Y 575.751,Z 685.03,A -85,B 0,C 180,E1 2220.129,E2 2220.129} C_VEL
LIN {X 0,Y 575.889,Z 685.03,A -85,B 0,C 180,E1 2225.209,E2 2225.209} C_VEL
LIN {X 0,Y 575.807,Z 685.088,A -85,B 0,C 180,E1 2228.603,E2 2228.603} C_VEL
LIN {X 0,Y 578.617,Z 700.562,A -85,B 0,C 180,E1 2229.072,E2 2229.072} C_VEL
LIN {X 0,Y 578.152,Z 734.556,A -85,B 0,C 180,E1 2230.311,E2 2230.311} C_VEL
LIN {X 0,Y 577.604,Z 765.923,A -85,B 0,C 180,E1 2232.108,E2 2232.108} C_VEL
LIN {X 0,Y 577.067,Z 794.367,A -85,B 0,C 180,E1 2234.45,E2 2234.45} C_VEL
LIN {X 0,Y 576.623,Z 817.829,A -85,B 0,C 180,E1 2237.144,E2 2237.144} C_VEL
LIN {X 0,Y 576.405,Z 836.743,A -85,B 0,C 180,E1 2240.2,E2 2240.2} C_VEL
LIN {X 0,Y 576.232,Z 849.504,A -85,B 0,C 180,E1 2243.23,E2 2243.23} C_VEL
LIN {X 0,Y 576.294,Z 857.203,A -85,B 0,C 180,E1 2246.244,E2 2246.244} C_VEL
LIN {X 0,Y 576.255,Z 859.949,A -85,B 0,C 180,E1 2248.497,E2 2248.497} C_VEL
LIN {X 0,Y 576.259,Z 859.892,A -85,B 0,C 180,E1 2251.498,E2 2251.498} C_VEL
LIN {X 0,Y 576.263,Z 855.514,A -85,B 0,C 180,E1 2254.504,E2 2254.504} C_VEL
LIN {X 0,Y 576.434,Z 845,A -85,B 0,C 180,E1 2257.898,E2 2257.898} C_VEL
LIN {X 0,Y 576.612,Z 828.684,A -85,B 0,C 180,E1 2261.149,E2 2261.149} C_VEL
LIN {X 0,Y 576.944,Z 806.981,A -85,B 0,C 180,E1 2264.119,E2 2264.119} C_VEL
LIN {X 0,Y 577.358,Z 780.446,A -85,B 0,C 180,E1 2266.707,E2 2266.707} C_VEL
LIN {X 0,Y 577.844,Z 750.836,A -85,B 0,C 180,E1 2268.754,E2 2268.754} C_VEL
LIN {X 0,Y 578.382,Z 718.914,A -85,B 0,C 180,E1 2270.253,E2 2270.253} C_VEL
LIN {X 0,Y 577.804,Z 691.288,A -85,B 0,C 180,E1 2271.099,E2 2271.099} C_VEL
LIN {X 0,Y 576.147,Z 685.03,A -85,B 0,C 180,E1 2271.313,E2 2271.313} C_VEL
LIN {X 0,Y 575.83,Z 685.03,A -85,B 0,C 180,E1 2278.144,E2 2278.144} C_VEL
LIN {X 0,Y 575.862,Z 685.03,A -85,B 0,C 180,E1 2283.386,E2 2283.386} C_VEL
LIN {X 0,Y 575.693,Z 685.03,A -85,B 0,C 180,E1 2288.982,E2 2288.982} C_VEL
LIN {X 0,Y 575.719,Z 685.03,A -85,B 0,C 180,E1 2295.047,E2 2295.047} C_VEL
LIN {X 0,Y 575.734,Z 685.03,A -85,B 0,C 180,E1 2301.029,E2 2301.029} C_VEL
LIN {X 0,Y 575.675,Z 685.03,A -85,B 0,C 180,E1 2306.608,E2 2306.608} C_VEL
LIN {X 0,Y 575.705,Z 685.03,A -85,B 0,C 180,E1 2311.855,E2 2311.855} C_VEL
LIN {X 0,Y 575.688,Z 685.03,A -85,B 0,C 180,E1 2316.853,E2 2316.853} C_VEL
LIN {X 0,Y 575.943,Z 685.03,A -85,B 0,C 180,E1 2321.68,E2 2321.68} C_VEL
LIN {X 0,Y 576.167,Z 685.03,A -85,B 0,C 180,E1 2326.371,E2 2326.371} C_VEL
LIN {X 0,Y 575.969,Z 685.03,A -85,B 0,C 180,E1 2332.701,E2 2332.701} C_VEL
LIN {X 0,Y 576.116,Z 685.03,A -85,B 0,C 180,E1 2337.001,E2 2337.001} C_VEL
LIN {X 0,Y 576.258,Z 685.03,A -85,B 0,C 180,E1 2341.504,E2 2341.504} C_VEL
LIN {X 0,Y 576.205,Z 685.03,A -85,B 0,C 180,E1 2346.016,E2 2346.016} C_VEL
LIN {X 0,Y 575.862,Z 685.03,A -85,B 0,C 180,E1 2349.172,E2 2349.172} C_VEL
LIN {X 0,Y 574.611,Z 685.03,A -85,B 0,C 180,E1 2350.033,E2 2350.033} C_VEL
LIN {X 0,Y 568.013,Z 685.03,A -85,B 0,C 180,E1 2352.373,E2 2352.373} C_VEL
LIN {X 0,Y 567.904,Z 685.03,A -85,B 0,C 180,E1 2352.594,E2 2352.594} C_VEL
LIN {X 0,Y 567.953,Z 685.03,A -85,B 0,C 180,E1 2356.995,E2 2356.995} C_VEL
LIN {X 0,Y 567.885,Z 685.03,A -85,B 0,C 180,E1 2361.841,E2 2361.841} C_VEL
LIN {X 0,Y 567.779,Z 685.03,A -85,B 0,C 180,E1 2366.861,E2 2366.861} C_VEL
LIN {X 0,Y 567.74,Z 685.03,A -85,B 0,C 180,E1 2372.113,E2 2372.113} C_VEL
LIN {X 0,Y 567.9,Z 685.03,A -85,B 0,C 180,E1 2377.673,E2 2377.673} C_VEL
LIN {X 0,Y 567.8,Z 685.03,A -85,B 0,C 180,E1 2383.708,E2 2383.708} C_VEL
LIN {X 0,Y 567.681,Z 685.03,A -85,B 0,C 180,E1 2388.353,E2 2388.353} C_VEL
LIN {X 0,Y 567.733,Z 685.03,A -85,B 0,C 180,E1 2394.216,E2 2394.216} C_VEL
LIN {X 0,Y 568.08,Z 685.217,A -85,B 0,C 180,E1 2397.854,E2 2397.854} C_VEL
LIN {X 0,Y 574.24,Z 699.905,A -85,B 0,C 180,E1 2398.451,E2 2398.451} C_VEL
LIN {X 0,Y 574.053,Z 773.551,A -85,B 0,C 180,E1 2399.606,E2 2399.606} C_VEL
LIN {X 0,Y 573.389,Z 810.746,A -85,B 0,C 180,E1 2400.743,E2 2400.743} C_VEL
LIN {X 0,Y 572.435,Z 846.852,A -85,B 0,C 180,E1 2402.422,E2 2402.422} C_VEL
LIN {X 0,Y 571.367,Z 882.128,A -85,B 0,C 180,E1 2404.703,E2 2404.703} C_VEL
LIN {X 0,Y 570.267,Z 914.657,A -85,B 0,C 180,E1 2407.5,E2 2407.5} C_VEL
LIN {X 0,Y 569.417,Z 943.702,A -85,B 0,C 180,E1 2410.777,E2 2410.777} C_VEL
LIN {X 0,Y 568.721,Z 968.095,A -85,B 0,C 180,E1 2414.418,E2 2414.418} C_VEL
LIN {X 0,Y 568.416,Z 986.457,A -85,B 0,C 180,E1 2418.129,E2 2418.129} C_VEL
LIN {X 0,Y 568.319,Z 999.72,A -85,B 0,C 180,E1 2421.989,E2 2421.989} C_VEL
LIN {X 0,Y 568.219,Z 1006.973,A -85,B 0,C 180,E1 2425.432,E2 2425.432} C_VEL
LIN {X 0,Y 568.252,Z 1010.098,A -85,B 0,C 180,E1 2428.481,E2 2428.481} C_VEL
LIN {X 0,Y 568.391,Z 1010.095,A -85,B 0,C 180,E1 2431.524,E2 2431.524} C_VEL
LIN {X 0,Y 568.362,Z 1005.383,A -85,B 0,C 180,E1 2435.53,E2 2435.53} C_VEL
LIN {X 0,Y 568.379,Z 995.076,A -85,B 0,C 180,E1 2439.554,E2 2439.554} C_VEL
LIN {X 0,Y 568.609,Z 979.449,A -85,B 0,C 180,E1 2443.43,E2 2443.43} C_VEL
LIN {X 0,Y 569.049,Z 958.14,A -85,B 0,C 180,E1 2447.192,E2 2447.192} C_VEL
LIN {X 0,Y 569.752,Z 932.862,A -85,B 0,C 180,E1 2450.548,E2 2450.548} C_VEL
LIN {X 0,Y 570.71,Z 901.953,A -85,B 0,C 180,E1 2453.686,E2 2453.686} C_VEL
LIN {X 0,Y 571.8,Z 867.688,A -85,B 0,C 180,E1 2456.32,E2 2456.32} C_VEL
LIN {X 0,Y 572.935,Z 830.849,A -85,B 0,C 180,E1 2458.398,E2 2458.398} C_VEL
LIN {X 0,Y 573.754,Z 792.513,A -85,B 0,C 180,E1 2459.886,E2 2459.886} C_VEL
LIN {X 0,Y 574.414,Z 754.188,A -85,B 0,C 180,E1 2460.753,E2 2460.753} C_VEL
LIN {X 0,Y 573.821,Z 698.739,A -85,B 0,C 180,E1 2461.591,E2 2461.591} C_VEL
LIN {X 0,Y 568.121,Z 685.03,A -85,B 0,C 180,E1 2462.18,E2 2462.18} C_VEL
LIN {X 0,Y 567.693,Z 685.03,A -85,B 0,C 180,E1 2467.694,E2 2467.694} C_VEL
LIN {X 0,Y 567.731,Z 685.03,A -85,B 0,C 180,E1 2473.721,E2 2473.721} C_VEL
LIN {X 0,Y 567.827,Z 685.03,A -85,B 0,C 180,E1 2478.365,E2 2478.365} C_VEL
LIN {X 0,Y 567.853,Z 685.03,A -85,B 0,C 180,E1 2484.223,E2 2484.223} C_VEL
LIN {X 0,Y 567.809,Z 685.03,A -85,B 0,C 180,E1 2489.671,E2 2489.671} C_VEL
LIN {X 0,Y 567.903,Z 685.03,A -85,B 0,C 180,E1 2494.839,E2 2494.839} C_VEL
LIN {X 0,Y 567.965,Z 685.03,A -85,B 0,C 180,E1 2499.793,E2 2499.793} C_VEL
LIN {X 0,Y 568.034,Z 685.03,A -85,B 0,C 180,E1 2503.685,E2 2503.685} C_VEL
LIN {X 0,Y 570.078,Z 699.718,A -85,B 0,C 180,E1 2503.936,E2 2503.936} C_VEL
LIN {X 0,Y 569.947,Z 743.94,A -85,B 0,C 180,E1 2504.645,E2 2504.645} C_VEL
LIN {X 0,Y 569.668,Z 772.355,A -85,B 0,C 180,E1 2505.715,E2 2505.715} C_VEL
LIN {X 0,Y 569.219,Z 798.664,A -85,B 0,C 180,E1 2507.364,E2 2507.364} C_VEL
LIN {X 0,Y 568.888,Z 821.169,A -85,B 0,C 180,E1 2509.49,E2 2509.49} C_VEL
LIN {X 0,Y 568.582,Z 839.018,A -85,B 0,C 180,E1 2511.988,E2 2511.988} C_VEL
LIN {X 0,Y 568.492,Z 850.535,A -85,B 0,C 180,E1 2514.428,E2 2514.428} C_VEL
LIN {X 0,Y 568.457,Z 857.612,A -85,B 0,C 180,E1 2516.954,E2 2516.954} C_VEL
LIN {X 0,Y 568.386,Z 860.455,A -85,B 0,C 180,E1 2519.997,E2 2519.997} C_VEL
LIN {X 0,Y 568.441,Z 857.444,A -85,B 0,C 180,E1 2523.04,E2 2523.04} C_VEL
LIN {X 0,Y 568.475,Z 849.168,A -85,B 0,C 180,E1 2525.825,E2 2525.825} C_VEL
LIN {X 0,Y 568.625,Z 835.009,A -85,B 0,C 180,E1 2528.581,E2 2528.581} C_VEL
LIN {X 0,Y 568.953,Z 817.018,A -85,B 0,C 180,E1 2530.877,E2 2530.877} C_VEL
LIN {X 0,Y 569.322,Z 793.68,A -85,B 0,C 180,E1 2532.918,E2 2532.918} C_VEL
LIN {X 0,Y 569.708,Z 767.858,A -85,B 0,C 180,E1 2534.409,E2 2534.409} C_VEL
LIN {X 0,Y 570.061,Z 738.78,A -85,B 0,C 180,E1 2535.393,E2 2535.393} C_VEL
LIN {X 0,Y 569.316,Z 690.477,A -85,B 0,C 180,E1 2536.115,E2 2536.115} C_VEL
LIN {X 0,Y 568.061,Z 685.03,A -85,B 0,C 180,E1 2536.27,E2 2536.27} C_VEL
LIN {X 0,Y 567.904,Z 685.03,A -85,B 0,C 180,E1 2541.833,E2 2541.833} C_VEL
LIN {X 0,Y 567.805,Z 685.03,A -85,B 0,C 180,E1 2546.852,E2 2546.852} C_VEL
LIN {X 0,Y 567.718,Z 685.03,A -85,B 0,C 180,E1 2552.107,E2 2552.107} C_VEL
LIN {X 0,Y 568.01,Z 685.03,A -85,B 0,C 180,E1 2557.656,E2 2557.656} C_VEL
LIN {X 0,Y 567.727,Z 685.03,A -85,B 0,C 180,E1 2564.133,E2 2564.133} C_VEL
LIN {X 0,Y 567.819,Z 685.03,A -85,B 0,C 180,E1 2568.359,E2 2568.359} C_VEL
LIN {X 0,Y 567.811,Z 685.03,A -85,B 0,C 180,E1 2574.216,E2 2574.216} C_VEL
LIN {X 0,Y 567.861,Z 685.03,A -85,B 0,C 180,E1 2579.671,E2 2579.671} C_VEL
LIN {X 0,Y 567.933,Z 685.03,A -85,B 0,C 180,E1 2584.838,E2 2584.838} C_VEL
LIN {X 0,Y 567.883,Z 685.03,A -85,B 0,C 180,E1 2588.282,E2 2588.282} C_VEL
LIN {X 0,Y 571.233,Z 700.747,A -85,B 0,C 180,E1 2588.795,E2 2588.795} C_VEL
LIN {X 0,Y 570.702,Z 734.549,A -85,B 0,C 180,E1 2590.043,E2 2590.043} C_VEL
LIN {X 0,Y 570.006,Z 765.8,A -85,B 0,C 180,E1 2591.853,E2 2591.853} C_VEL
LIN {X 0,Y 569.351,Z 794.36,A -85,B 0,C 180,E1 2594.233,E2 2594.233} C_VEL
LIN {X 0,Y 568.844,Z 817.821,A -85,B 0,C 180,E1 2596.966,E2 2596.966} C_VEL
LIN {X 0,Y 568.537,Z 836.742,A -85,B 0,C 180,E1 2600.063,E2 2600.063} C_VEL
LIN {X 0,Y 568.353,Z 849.5,A -85,B 0,C 180,E1 2603.135,E2 2603.135} C_VEL
LIN {X 0,Y 568.402,Z 857.202,A -85,B 0,C 180,E1 2606.192,E2 2606.192} C_VEL
LIN {X 0,Y 568.371,Z 859.949,A -85,B 0,C 180,E1 2608.476,E2 2608.476} C_VEL
LIN {X 0,Y 568.375,Z 859.892,A -85,B 0,C 180,E1 2611.519,E2 2611.519} C_VEL
LIN {X 0,Y 568.414,Z 854.24,A -85,B 0,C 180,E1 2615.111,E2 2615.111} C_VEL
LIN {X 0,Y 568.539,Z 843.475,A -85,B 0,C 180,E1 2618.392,E2 2618.392} C_VEL
LIN {X 0,Y 568.809,Z 826.122,A -85,B 0,C 180,E1 2621.72,E2 2621.72} C_VEL
LIN {X 0,Y 569.177,Z 803.831,A -85,B 0,C 180,E1 2624.675,E2 2624.675} C_VEL
LIN {X 0,Y 569.743,Z 777.368,A -85,B 0,C 180,E1 2627.187,E2 2627.187} C_VEL
LIN {X 0,Y 570.421,Z 747.419,A -85,B 0,C 180,E1 2629.208,E2 2629.208} C_VEL
LIN {X 0,Y 571.056,Z 715.869,A -85,B 0,C 180,E1 2630.639,E2 2630.639} C_VEL
LIN {X 0,Y 570.405,Z 692.987,A -85,B 0,C 180,E1 2631.348,E2 2631.348} C_VEL
LIN {X 0,Y 568.211,Z 685.03,A -85,B 0,C 180,E1 2631.665,E2 2631.665} C_VEL
LIN {X 0,Y 567.84,Z 685.03,A -85,B 0,C 180,E1 2638.576,E2 2638.576} C_VEL
LIN {X 0,Y 567.783,Z 685.03,A -85,B 0,C 180,E1 2644.537,E2 2644.537} C_VEL
LIN {X 0,Y 567.756,Z 685.03,A -85,B 0,C 180,E1 2649.633,E2 2649.633} C_VEL
LIN {X 0,Y 567.756,Z 685.03,A -85,B 0,C 180,E1 2655.858,E2 2655.858} C_VEL
LIN {X 0,Y 567.822,Z 685.03,A -85,B 0,C 180,E1 2660.415,E2 2660.415} C_VEL
LIN {X 0,Y 567.728,Z 685.03,A -85,B 0,C 180,E1 2665.484,E2 2665.484} C_VEL
LIN {X 0,Y 567.823,Z 685.03,A -85,B 0,C 180,E1 2669.68,E2 2669.68} C_VEL
LIN {X 0,Y 567.89,Z 685.03,A -85,B 0,C 180,E1 2674.846,E2 2674.846} C_VEL
LIN {X 0,Y 568.038,Z 685.03,A -85,B 0,C 180,E1 2679.802,E2 2679.802} C_VEL
LIN {X 0,Y 568.244,Z 685.03,A -85,B 0,C 180,E1 2686.177,E2 2686.177} C_VEL
LIN {X 0,Y 568.045,Z 685.03,A -85,B 0,C 180,E1 2692.689,E2 2692.689} C_VEL
LIN {X 0,Y 568.211,Z 685.03,A -85,B 0,C 180,E1 2696.959,E2 2696.959} C_VEL
LIN {X 0,Y 568.371,Z 685.03,A -85,B 0,C 180,E1 2701.525,E2 2701.525} C_VEL
LIN {X 0,Y 568.272,Z 685.03,A -85,B 0,C 180,E1 2706.1,E2 2706.1} C_VEL
LIN {X 0,Y 567.941,Z 685.03,A -85,B 0,C 180,E1 2712.275,E2 2712.275} C_VEL
LIN {X 0,Y 567.904,Z 685.03,A -85,B 0,C 180,E1 2712.594,E2 2712.594} C_VEL
LIN {X 0,Y 563.97,Z 685.03,A -85,B 0,C 180,E1 2714.316,E2 2714.316} C_VEL
LIN {X 0,Y 560.013,Z 685.03,A -85,B 0,C 180,E1 2716.061,E2 2716.061} C_VEL
LIN {X 0,Y 559.933,Z 685.03,A -85,B 0,C 180,E1 2722.168,E2 2722.168} C_VEL
LIN {X 0,Y 559.825,Z 685.03,A -85,B 0,C 180,E1 2727.274,E2 2727.274} C_VEL
LIN {X 0,Y 559.764,Z 685.03,A -85,B 0,C 180,E1 2732.627,E2 2732.627} C_VEL
LIN {X 0,Y 559.907,Z 685.03,A -85,B 0,C 180,E1 2738.307,E2 2738.307} C_VEL
LIN {X 0,Y 559.859,Z 685.03,A -85,B 0,C 180,E1 2743.303,E2 2743.303} C_VEL
LIN {X 0,Y 559.759,Z 685.03,A -85,B 0,C 180,E1 2749.01,E2 2749.01} C_VEL
LIN {X 0,Y 559.944,Z 685.03,A -85,B 0,C 180,E1 2755.534,E2 2755.534} C_VEL
LIN {X 0,Y 560.184,Z 685.07,A -85,B 0,C 180,E1 2757.343,E2 2757.343} C_VEL
LIN {X 0,Y 567.58,Z 703.599,A -85,B 0,C 180,E1 2758.091,E2 2758.091} C_VEL
LIN {X 0,Y 567.21,Z 775.295,A -85,B 0,C 180,E1 2759.243,E2 2759.243} C_VEL
LIN {X 0,Y 566.366,Z 814.421,A -85,B 0,C 180,E1 2760.492,E2 2760.492} C_VEL
LIN {X 0,Y 565.164,Z 852.295,A -85,B 0,C 180,E1 2762.352,E2 2762.352} C_VEL
LIN {X 0,Y 563.807,Z 887.863,A -85,B 0,C 180,E1 2764.789,E2 2764.789} C_VEL
LIN {X 0,Y 562.596,Z 920.138,A -85,B 0,C 180,E1 2767.744,E2 2767.744} C_VEL
LIN {X 0,Y 561.596,Z 947.704,A -85,B 0,C 180,E1 2771.047,E2 2771.047} C_VEL
LIN {X 0,Y 560.91,Z 971.005,A -85,B 0,C 180,E1 2774.726,E2 2774.726} C_VEL
LIN {X 0,Y 560.533,Z 988.007,A -85,B 0,C 180,E1 2778.353,E2 2778.353} C_VEL
LIN {X 0,Y 560.458,Z 999.719,A -85,B 0,C 180,E1 2781.876,E2 2781.876} C_VEL
LIN {X 0,Y 560.321,Z 1006.976,A -85,B 0,C 180,E1 2785.368,E2 2785.368} C_VEL
LIN {X 0,Y 560.349,Z 1010.1,A -85,B 0,C 180,E1 2788.459,E2 2788.459} C_VEL
LIN {X 0,Y 560.485,Z 1010.097,A -85,B 0,C 180,E1 2791.545,E2 2791.545} C_VEL
LIN {X 0,Y 560.464,Z 1005.826,A -85,B 0,C 180,E1 2795.364,E2 2795.364} C_VEL
LIN {X 0,Y 560.523,Z 996.312,A -85,B 0,C 180,E1 2799.298,E2 2799.298} C_VEL
LIN {X 0,Y 560.783,Z 981.284,A -85,B 0,C 180,E1 2803.225,E2 2803.225} C_VEL
LIN {X 0,Y 561.22,Z 960.914,A -85,B 0,C 180,E1 2807.005,E2 2807.005} C_VEL
LIN {X 0,Y 562.085,Z 934.606,A -85,B 0,C 180,E1 2810.635,E2 2810.635} C_VEL
LIN {X 0,Y 563.191,Z 903.979,A -85,B 0,C 180,E1 2813.835,E2 2813.835} C_VEL
LIN {X 0,Y 564.48,Z 869.579,A -85,B 0,C 180,E1 2816.555,E2 2816.555} C_VEL
LIN {X 0,Y 565.76,Z 834.438,A -85,B 0,C 180,E1 2818.607,E2 2818.607} C_VEL
LIN {X 0,Y 566.754,Z 797.129,A -85,B 0,C 180,E1 2820.137,E2 2820.137} C_VEL
LIN {X 0,Y 567.557,Z 761.837,A -85,B 0,C 180,E1 2821.035,E2 2821.035} C_VEL
LIN {X 0,Y 567.038,Z 701.246,A -85,B 0,C 180,E1 2821.977,E2 2821.977} C_VEL
LIN {X 0,Y 560.213,Z 685.03,A -85,B 0,C 180,E1 2822.695,E2 2822.695} C_VEL
LIN {X 0,Y 559.74,Z 685.03,A -85,B 0,C 180,E1 2828.574,E2 2828.574} C_VEL
LIN {X 0,Y 559.817,Z 685.03,A -85,B 0,C 180,E1 2834.5,E2 2834.5} C_VEL
LIN {X 0,Y 559.846,Z 685.03,A -85,B 0,C 180,E1 2839.692,E2 2839.692} C_VEL
LIN {X 0,Y 559.838,Z 685.03,A -85,B 0,C 180,E1 2845.525,E2 2845.525} C_VEL
LIN {X 0,Y 559.841,Z 685.03,A -85,B 0,C 180,E1 2850.975,E2 2850.975} C_VEL
LIN {X 0,Y 559.925,Z 685.03,A -85,B 0,C 180,E1 2856.404,E2 2856.404} C_VEL
LIN {X 0,Y 559.965,Z 685.03,A -85,B 0,C 180,E1 2861.131,E2 2861.131} C_VEL
LIN {X 0,Y 560.141,Z 685.03,A -85,B 0,C 180,E1 2863.445,E2 2863.445} C_VEL
LIN {X 0,Y 562.484,Z 699.355,A -85,B 0,C 180,E1 2863.709,E2 2863.709} C_VEL
LIN {X 0,Y 562.342,Z 743.883,A -85,B 0,C 180,E1 2864.432,E2 2864.432} C_VEL
LIN {X 0,Y 561.984,Z 772.279,A -85,B 0,C 180,E1 2865.512,E2 2865.512} C_VEL
LIN {X 0,Y 561.468,Z 798.64,A -85,B 0,C 180,E1 2867.187,E2 2867.187} C_VEL
LIN {X 0,Y 561.067,Z 821.155,A -85,B 0,C 180,E1 2869.342,E2 2869.342} C_VEL
LIN {X 0,Y 560.727,Z 839.004,A -85,B 0,C 180,E1 2871.875,E2 2871.875} C_VEL
LIN {X 0,Y 560.577,Z 851.522,A -85,B 0,C 180,E1 2874.632,E2 2874.632} C_VEL
LIN {X 0,Y 560.574,Z 858.849,A -85,B 0,C 180,E1 2877.683,E2 2877.683} C_VEL
LIN {X 0,Y 560.486,Z 860.447,A -85,B 0,C 180,E1 2879.997,E2 2879.997} C_VEL
LIN {X 0,Y 560.542,Z 857.448,A -85,B 0,C 180,E1 2883.083,E2 2883.083} C_VEL
LIN {X 0,Y 560.583,Z 849.583,A -85,B 0,C 180,E1 2885.802,E2 2885.802} C_VEL
LIN {X 0,Y 560.774,Z 835.014,A -85,B 0,C 180,E1 2888.702,E2 2888.702} C_VEL
LIN {X 0,Y 561.129,Z 817.074,A -85,B 0,C 180,E1 2891.024,E2 2891.024} C_VEL
LIN {X 0,Y 561.559,Z 793.683,A -85,B 0,C 180,E1 2893.1,E2 2893.1} C_VEL
LIN {X 0,Y 562.03,Z 767.762,A -85,B 0,C 180,E1 2894.614,E2 2894.614} C_VEL
LIN {X 0,Y 562.446,Z 738.904,A -85,B 0,C 180,E1 2895.603,E2 2895.603} C_VEL
LIN {X 0,Y 561.672,Z 691.792,A -85,B 0,C 180,E1 2896.324,E2 2896.324} C_VEL
LIN {X 0,Y 560.138,Z 685.03,A -85,B 0,C 180,E1 2896.544,E2 2896.544} C_VEL
LIN {X 0,Y 559.953,Z 685.03,A -85,B 0,C 180,E1 2902.16,E2 2902.16} C_VEL
LIN {X 0,Y 559.84,Z 685.03,A -85,B 0,C 180,E1 2907.266,E2 2907.266} C_VEL
LIN {X 0,Y 559.742,Z 685.03,A -85,B 0,C 180,E1 2912.62,E2 2912.62} C_VEL
LIN {X 0,Y 559.99,Z 685.03,A -85,B 0,C 180,E1 2918.292,E2 2918.292} C_VEL
LIN {X 0,Y 559.797,Z 685.03,A -85,B 0,C 180,E1 2924.486,E2 2924.486} C_VEL
LIN {X 0,Y 559.831,Z 685.03,A -85,B 0,C 180,E1 2929.685,E2 2929.685} C_VEL
LIN {X 0,Y 559.811,Z 685.03,A -85,B 0,C 180,E1 2935.519,E2 2935.519} C_VEL
LIN {X 0,Y 559.888,Z 685.03,A -85,B 0,C 180,E1 2940.974,E2 2940.974} C_VEL
LIN {X 0,Y 559.984,Z 685.03,A -85,B 0,C 180,E1 2946.358,E2 2946.358} C_VEL
LIN {X 0,Y 559.956,Z 685.043,A -85,B 0,C 180,E1 2947.967,E2 2947.967} C_VEL
LIN {X 0,Y 563.86,Z 701.81,A -85,B 0,C 180,E1 2948.534,E2 2948.534} C_VEL
LIN {X 0,Y 563.217,Z 735.005,A -85,B 0,C 180,E1 2949.79,E2 2949.79} C_VEL
LIN {X 0,Y 562.449,Z 765.382,A -85,B 0,C 180,E1 2951.57,E2 2951.57} C_VEL
LIN {X 0,Y 561.704,Z 793.327,A -85,B 0,C 180,E1 2953.913,E2 2953.913} C_VEL
LIN {X 0,Y 561.125,Z 816.381,A -85,B 0,C 180,E1 2956.585,E2 2956.585} C_VEL
LIN {X 0,Y 560.749,Z 834.784,A -85,B 0,C 180,E1 2959.531,E2 2959.531} C_VEL
LIN {X 0,Y 560.569,Z 848.177,A -85,B 0,C 180,E1 2962.651,E2 2962.651} C_VEL
LIN {X 0,Y 560.515,Z 857.201,A -85,B 0,C 180,E1 2966.138,E2 2966.138} C_VEL
LIN {X 0,Y 560.467,Z 859.949,A -85,B 0,C 180,E1 2968.455,E2 2968.455} C_VEL
LIN {X 0,Y 560.471,Z 859.892,A -85,B 0,C 180,E1 2971.541,E2 2971.541} C_VEL
LIN {X 0,Y 560.522,Z 854.292,A -85,B 0,C 180,E1 2975.162,E2 2975.162} C_VEL
LIN {X 0,Y 560.652,Z 843.479,A -85,B 0,C 180,E1 2978.511,E2 2978.511} C_VEL
LIN {X 0,Y 560.942,Z 826.446,A -85,B 0,C 180,E1 2981.835,E2 2981.835} C_VEL
LIN {X 0,Y 561.41,Z 804.922,A -85,B 0,C 180,E1 2984.757,E2 2984.757} C_VEL
LIN {X 0,Y 562.089,Z 778.93,A -85,B 0,C 180,E1 2987.301,E2 2987.301} C_VEL
LIN {X 0,Y 562.835,Z 749.187,A -85,B 0,C 180,E1 2989.376,E2 2989.376} C_VEL
LIN {X 0,Y 563.633,Z 716.649,A -85,B 0,C 180,E1 2990.895,E2 2990.895} C_VEL
LIN {X 0,Y 563.09,Z 694.986,A -85,B 0,C 180,E1 2991.593,E2 2991.593} C_VEL
LIN {X 0,Y 560.27,Z 685.03,A -85,B 0,C 180,E1 2991.944,E2 2991.944} C_VEL
LIN {X 0,Y 559.923,Z 685.03,A -85,B 0,C 180,E1 2997.267,E2 2997.267} C_VEL
LIN {X 0,Y 559.899,Z 685.03,A -85,B 0,C 180,E1 3003.347,E2 3003.347} C_VEL
LIN {X 0,Y 559.758,Z 685.03,A -85,B 0,C 180,E1 3008.587,E2 3008.587} C_VEL
LIN {X 0,Y 559.779,Z 685.03,A -85,B 0,C 180,E1 3014.498,E2 3014.498} C_VEL
LIN {X 0,Y 559.844,Z 685.03,A -85,B 0,C 180,E1 3019.701,E2 3019.701} C_VEL
LIN {X 0,Y 559.845,Z 685.03,A -85,B 0,C 180,E1 3025.534,E2 3025.534} C_VEL
LIN {X 0,Y 559.853,Z 685.03,A -85,B 0,C 180,E1 3030.983,E2 3030.983} C_VEL
LIN {X 0,Y 559.9,Z 685.03,A -85,B 0,C 180,E1 3036.398,E2 3036.398} C_VEL
LIN {X 0,Y 560.124,Z 685.03,A -85,B 0,C 180,E1 3041.144,E2 3041.144} C_VEL
LIN {X 0,Y 560.295,Z 685.03,A -85,B 0,C 180,E1 3045.977,E2 3045.977} C_VEL
LIN {X 0,Y 560.22,Z 685.03,A -85,B 0,C 180,E1 3052.264,E2 3052.264} C_VEL
LIN {X 0,Y 560.302,Z 685.03,A -85,B 0,C 180,E1 3056.916,E2 3056.916} C_VEL
LIN {X 0,Y 560.459,Z 685.03,A -85,B 0,C 180,E1 3061.546,E2 3061.546} C_VEL
LIN {X 0,Y 560.361,Z 685.03,A -85,B 0,C 180,E1 3066.187,E2 3066.187} C_VEL
LIN {X 0,Y 560.003,Z 685.03,A -85,B 0,C 180,E1 3072.585,E2 3072.585} C_VEL
LIN {X 0,Y 560.013,Z 685.03,A -85,B 0,C 180,E1 3076.061,E2 3076.061} C_VEL
LIN {X 0,Y 556.024,Z 685.03,A -85,B 0,C 180,E1 3077.805,E2 3077.805} C_VEL
LIN {X 0,Y 552.033,Z 685.03,A -85,B 0,C 180,E1 3079.574,E2 3079.574} C_VEL
LIN {X 0,Y 552.015,Z 685.03,A -85,B 0,C 180,E1 3085.564,E2 3085.564} C_VEL
LIN {X 0,Y 551.89,Z 685.03,A -85,B 0,C 180,E1 3091.3,E2 3091.3} C_VEL
LIN {X 0,Y 551.971,Z 685.03,A -85,B 0,C 180,E1 3097.551,E2 3097.551} C_VEL
LIN {X 0,Y 551.97,Z 685.03,A -85,B 0,C 180,E1 3103.115,E2 3103.115} C_VEL
LIN {X 0,Y 551.877,Z 685.03,A -85,B 0,C 180,E1 3108.987,E2 3108.987} C_VEL
LIN {X 0,Y 551.987,Z 685.03,A -85,B 0,C 180,E1 3115.097,E2 3115.097} C_VEL
LIN {X 0,Y 552.216,Z 685.299,A -85,B 0,C 180,E1 3116.815,E2 3116.815} C_VEL
LIN {X 0,Y 560.895,Z 706.692,A -85,B 0,C 180,E1 3117.711,E2 3117.711} C_VEL
LIN {X 0,Y 560.399,Z 775.282,A -85,B 0,C 180,E1 3118.827,E2 3118.827} C_VEL
LIN {X 0,Y 559.43,Z 814.304,A -85,B 0,C 180,E1 3120.084,E2 3120.084} C_VEL
LIN {X 0,Y 558.025,Z 852.134,A -85,B 0,C 180,E1 3121.957,E2 3121.957} C_VEL
LIN {X 0,Y 556.493,Z 887.574,A -85,B 0,C 180,E1 3124.41,E2 3124.41} C_VEL
LIN {X 0,Y 555.081,Z 920.284,A -85,B 0,C 180,E1 3127.442,E2 3127.442} C_VEL
LIN {X 0,Y 553.862,Z 948.743,A -85,B 0,C 180,E1 3130.918,E2 3130.918} C_VEL
LIN {X 0,Y 553.088,Z 970.827,A -85,B 0,C 180,E1 3134.471,E2 3134.471} C_VEL
LIN {X 0,Y 552.669,Z 988.01,A -85,B 0,C 180,E1 3138.185,E2 3138.185} C_VEL
LIN {X 0,Y 552.538,Z 1000.706,A -85,B 0,C 180,E1 3142.154,E2 3142.154} C_VEL
LIN {X 0,Y 552.452,Z 1006.978,A -85,B 0,C 180,E1 3145.302,E2 3145.302} C_VEL
LIN {X 0,Y 552.453,Z 1010.102,A -85,B 0,C 180,E1 3148.437,E2 3148.437} C_VEL
LIN {X 0,Y 552.579,Z 1010.099,A -85,B 0,C 180,E1 3151.567,E2 3151.567} C_VEL
LIN {X 0,Y 552.552,Z 1005.745,A -85,B 0,C 180,E1 3155.488,E2 3155.488} C_VEL
LIN {X 0,Y 552.625,Z 996.315,A -85,B 0,C 180,E1 3159.433,E2 3159.433} C_VEL
LIN {X 0,Y 552.929,Z 981.287,A -85,B 0,C 180,E1 3163.416,E2 3163.416} C_VEL
LIN {X 0,Y 553.485,Z 959.949,A -85,B 0,C 180,E1 3167.407,E2 3167.407} C_VEL
LIN {X 0,Y 554.483,Z 934.604,A -85,B 0,C 180,E1 3170.931,E2 3170.931} C_VEL
LIN {X 0,Y 555.801,Z 903.984,A -85,B 0,C 180,E1 3174.172,E2 3174.172} C_VEL
LIN {X 0,Y 557.249,Z 869.719,A -85,B 0,C 180,E1 3176.917,E2 3176.917} C_VEL
LIN {X 0,Y 558.735,Z 834.692,A -85,B 0,C 180,E1 3178.987,E2 3178.987} C_VEL
LIN {X 0,Y 559.866,Z 798.428,A -85,B 0,C 180,E1 3180.502,E2 3180.502} C_VEL
LIN {X 0,Y 560.791,Z 761.838,A -85,B 0,C 180,E1 3181.452,E2 3181.452} C_VEL
LIN {X 0,Y 560.344,Z 703.681,A -85,B 0,C 180,E1 3182.369,E2 3182.369} C_VEL
LIN {X 0,Y 552.242,Z 685.03,A -85,B 0,C 180,E1 3183.204,E2 3183.204} C_VEL
LIN {X 0,Y 551.833,Z 685.03,A -85,B 0,C 180,E1 3190.034,E2 3190.034} C_VEL
LIN {X 0,Y 551.943,Z 685.03,A -85,B 0,C 180,E1 3195.309,E2 3195.309} C_VEL
LIN {X 0,Y 551.966,Z 685.03,A -85,B 0,C 180,E1 3201.039,E2 3201.039} C_VEL
LIN {X 0,Y 551.881,Z 685.03,A -85,B 0,C 180,E1 3206.847,E2 3206.847} C_VEL
LIN {X 0,Y 551.913,Z 685.03,A -85,B 0,C 180,E1 3212.301,E2 3212.301} C_VEL
LIN {X 0,Y 552.016,Z 685.03,A -85,B 0,C 180,E1 3217.497,E2 3217.497} C_VEL
LIN {X 0,Y 552.204,Z 685.03,A -85,B 0,C 180,E1 3223.204,E2 3223.204} C_VEL
LIN {X 0,Y 554.93,Z 699.559,A -85,B 0,C 180,E1 3223.484,E2 3223.484} C_VEL
LIN {X 0,Y 554.728,Z 743.827,A -85,B 0,C 180,E1 3224.213,E2 3224.213} C_VEL
LIN {X 0,Y 554.282,Z 772.077,A -85,B 0,C 180,E1 3225.297,E2 3225.297} C_VEL
LIN {X 0,Y 553.687,Z 798.616,A -85,B 0,C 180,E1 3227.004,E2 3227.004} C_VEL
LIN {X 0,Y 553.285,Z 820.363,A -85,B 0,C 180,E1 3229.094,E2 3229.094} C_VEL
LIN {X 0,Y 552.89,Z 838.99,A -85,B 0,C 180,E1 3231.759,E2 3231.759} C_VEL
LIN {X 0,Y 552.72,Z 850.686,A -85,B 0,C 180,E1 3234.311,E2 3234.311} C_VEL
LIN {X 0,Y 552.683,Z 857.615,A -85,B 0,C 180,E1 3236.867,E2 3236.867} C_VEL
LIN {X 0,Y 552.587,Z 860.438,A -85,B 0,C 180,E1 3239.997,E2 3239.997} C_VEL
LIN {X 0,Y 552.669,Z 857.452,A -85,B 0,C 180,E1 3243.127,E2 3243.127} C_VEL
LIN {X 0,Y 552.702,Z 849.103,A -85,B 0,C 180,E1 3246.006,E2 3246.006} C_VEL
LIN {X 0,Y 552.926,Z 835.019,A -85,B 0,C 180,E1 3248.826,E2 3248.826} C_VEL
LIN {X 0,Y 553.317,Z 816.897,A -85,B 0,C 180,E1 3251.2,E2 3251.2} C_VEL
LIN {X 0,Y 553.833,Z 793.677,A -85,B 0,C 180,E1 3253.286,E2 3253.286} C_VEL
LIN {X 0,Y 554.352,Z 768.32,A -85,B 0,C 180,E1 3254.795,E2 3254.795} C_VEL
LIN {X 0,Y 554.846,Z 739.381,A -85,B 0,C 180,E1 3255.81,E2 3255.81} C_VEL
LIN {X 0,Y 554.188,Z 693.466,A -85,B 0,C 180,E1 3256.529,E2 3256.529} C_VEL
LIN {X 0,Y 552.217,Z 685.03,A -85,B 0,C 180,E1 3256.763,E2 3256.763} C_VEL
LIN {X 0,Y 552.018,Z 685.03,A -85,B 0,C 180,E1 3262.496,E2 3262.496} C_VEL
LIN {X 0,Y 551.884,Z 685.03,A -85,B 0,C 180,E1 3267.692,E2 3267.692} C_VEL
LIN {X 0,Y 551.834,Z 685.03,A -85,B 0,C 180,E1 3273.147,E2 3273.147} C_VEL
LIN {X 0,Y 552.01,Z 685.03,A -85,B 0,C 180,E1 3278.949,E2 3278.949} C_VEL
LIN {X 0,Y 551.917,Z 685.03,A -85,B 0,C 180,E1 3285.296,E2 3285.296} C_VEL
LIN {X 0,Y 551.949,Z 685.03,A -85,B 0,C 180,E1 3291.032,E2 3291.032} C_VEL
LIN {X 0,Y 551.903,Z 685.03,A -85,B 0,C 180,E1 3296.845,E2 3296.845} C_VEL
LIN {X 0,Y 551.984,Z 685.03,A -85,B 0,C 180,E1 3302.302,E2 3302.302} C_VEL
LIN {X 0,Y 552.021,Z 685.169,A -85,B 0,C 180,E1 3307.636,E2 3307.636} C_VEL
LIN {X 0,Y 556.483,Z 703.564,A -85,B 0,C 180,E1 3308.286,E2 3308.286} C_VEL
LIN {X 0,Y 555.722,Z 736.176,A -85,B 0,C 180,E1 3309.565,E2 3309.565} C_VEL
LIN {X 0,Y 554.829,Z 766.79,A -85,B 0,C 180,E1 3311.414,E2 3311.414} C_VEL
LIN {X 0,Y 553.983,Z 794.345,A -85,B 0,C 180,E1 3313.784,E2 3313.784} C_VEL
LIN {X 0,Y 553.291,Z 817.805,A -85,B 0,C 180,E1 3316.592,E2 3316.592} C_VEL
LIN {X 0,Y 552.875,Z 836.054,A -85,B 0,C 180,E1 3319.638,E2 3319.638} C_VEL
LIN {X 0,Y 552.634,Z 849.494,A -85,B 0,C 180,E1 3322.939,E2 3322.939} C_VEL
LIN {X 0,Y 552.628,Z 857.2,A -85,B 0,C 180,E1 3326.083,E2 3326.083} C_VEL
LIN {X 0,Y 552.563,Z 859.948,A -85,B 0,C 180,E1 3328.433,E2 3328.433} C_VEL
LIN {X 0,Y 552.568,Z 859.893,A -85,B 0,C 180,E1 3331.563,E2 3331.563} C_VEL
LIN {X 0,Y 552.62,Z 854.293,A -85,B 0,C 180,E1 3335.236,E2 3335.236} C_VEL
LIN {X 0,Y 552.788,Z 843.483,A -85,B 0,C 180,E1 3338.633,E2 3338.633} C_VEL
LIN {X 0,Y 553.085,Z 826.453,A -85,B 0,C 180,E1 3342.005,E2 3342.005} C_VEL
LIN {X 0,Y 553.659,Z 804.861,A -85,B 0,C 180,E1 3344.976,E2 3344.976} C_VEL
LIN {X 0,Y 554.443,Z 778.347,A -85,B 0,C 180,E1 3347.597,E2 3347.597} C_VEL
LIN {X 0,Y 555.338,Z 749.057,A -85,B 0,C 180,E1 3349.657,E2 3349.657} C_VEL
LIN {X 0,Y 556.243,Z 716.897,A -85,B 0,C 180,E1 3351.176,E2 3351.176} C_VEL
LIN {X 0,Y 555.649,Z 696.561,A -85,B 0,C 180,E1 3351.856,E2 3351.856} C_VEL
LIN {X 0,Y 552.278,Z 685.03,A -85,B 0,C 180,E1 3352.304,E2 3352.304} C_VEL
LIN {X 0,Y 552.004,Z 685.03,A -85,B 0,C 180,E1 3358.998,E2 3358.998} C_VEL
LIN {X 0,Y 551.932,Z 685.03,A -85,B 0,C 180,E1 3365.039,E2 3365.039} C_VEL
LIN {X 0,Y 551.866,Z 685.03,A -85,B 0,C 180,E1 3371.014,E2 3371.014} C_VEL
LIN {X 0,Y 551.94,Z 685.03,A -85,B 0,C 180,E1 3376.892,E2 3376.892} C_VEL
LIN {X 0,Y 551.962,Z 685.03,A -85,B 0,C 180,E1 3383.034,E2 3383.034} C_VEL
LIN {X 0,Y 551.919,Z 685.03,A -85,B 0,C 180,E1 3388.71,E2 3388.71} C_VEL
LIN {X 0,Y 552.075,Z 685.03,A -85,B 0,C 180,E1 3394.423,E2 3394.423} C_VEL
LIN {X 0,Y 552.212,Z 685.03,A -85,B 0,C 180,E1 3400.863,E2 3400.863} C_VEL
LIN {X 0,Y 552.379,Z 685.03,A -85,B 0,C 180,E1 3405.772,E2 3405.772} C_VEL
LIN {X 0,Y 552.306,Z 685.03,A -85,B 0,C 180,E1 3412.153,E2 3412.153} C_VEL
LIN {X 0,Y 552.403,Z 685.03,A -85,B 0,C 180,E1 3416.872,E2 3416.872} C_VEL
LIN {X 0,Y 552.55,Z 685.03,A -85,B 0,C 180,E1 3421.568,E2 3421.568} C_VEL
LIN {X 0,Y 552.43,Z 685.03,A -85,B 0,C 180,E1 3426.276,E2 3426.276} C_VEL
LIN {X 0,Y 552.108,Z 685.03,A -85,B 0,C 180,E1 3432.632,E2 3432.632} C_VEL
LIN {X 0,Y 552.103,Z 685.03,A -85,B 0,C 180,E1 3437.499,E2 3437.499} C_VEL
LIN {X 0,Y 552.033,Z 685.03,A -85,B 0,C 180,E1 3439.574,E2 3439.574} C_VEL
LIN {X 0,Y 548.023,Z 685.03,A -85,B 0,C 180,E1 3441.344,E2 3441.344} C_VEL
LIN {X 0,Y 544.025,Z 685.03,A -85,B 0,C 180,E1 3443.139,E2 3443.139} C_VEL
LIN {X 0,Y 543.955,Z 685.03,A -85,B 0,C 180,E1 3448.14,E2 3448.14} C_VEL
LIN {X 0,Y 543.927,Z 685.03,A -85,B 0,C 180,E1 3453.702,E2 3453.702} C_VEL
LIN {X 0,Y 544.028,Z 685.03,A -85,B 0,C 180,E1 3459.641,E2 3459.641} C_VEL
LIN {X 0,Y 544.014,Z 685.03,A -85,B 0,C 180,E1 3463.904,E2 3463.904} C_VEL
LIN {X 0,Y 543.921,Z 685.03,A -85,B 0,C 180,E1 3470.351,E2 3470.351} C_VEL
LIN {X 0,Y 544.23,Z 685.03,A -85,B 0,C 180,E1 3476.221,E2 3476.221} C_VEL
LIN {X 0,Y 554.204,Z 707.448,A -85,B 0,C 180,E1 3477.284,E2 3477.284} C_VEL
LIN {X 0,Y 553.626,Z 775.135,A -85,B 0,C 180,E1 3478.399,E2 3478.399} C_VEL
LIN {X 0,Y 552.503,Z 814.417,A -85,B 0,C 180,E1 3479.675,E2 3479.675} C_VEL
LIN {X 0,Y 550.942,Z 851.901,A -85,B 0,C 180,E1 3481.55,E2 3481.55} C_VEL
LIN {X 0,Y 549.147,Z 888.347,A -85,B 0,C 180,E1 3484.108,E2 3484.108} C_VEL
LIN {X 0,Y 547.544,Z 920.093,A -85,B 0,C 180,E1 3487.092,E2 3487.092} C_VEL
LIN {X 0,Y 546.232,Z 947.367,A -85,B 0,C 180,E1 3490.443,E2 3490.443} C_VEL
LIN {X 0,Y 545.29,Z 970.296,A -85,B 0,C 180,E1 3494.142,E2 3494.142} C_VEL
LIN {X 0,Y 544.828,Z 988.014,A -85,B 0,C 180,E1 3498.013,E2 3498.013} C_VEL
LIN {X 0,Y 544.714,Z 999.718,A -85,B 0,C 180,E1 3501.639,E2 3501.639} C_VEL
LIN {X 0,Y 544.552,Z 1006.981,A -85,B 0,C 180,E1 3505.234,E2 3505.234} C_VEL
LIN {X 0,Y 544.551,Z 1010.104,A -85,B 0,C 180,E1 3508.414,E2 3508.414} C_VEL
LIN {X 0,Y 544.673,Z 1010.101,A -85,B 0,C 180,E1 3511.59,E2 3511.59} C_VEL
LIN {X 0,Y 544.654,Z 1005.744,A -85,B 0,C 180,E1 3515.567,E2 3515.567} C_VEL
LIN {X 0,Y 544.726,Z 996.317,A -85,B 0,C 180,E1 3519.571,E2 3519.571} C_VEL
LIN {X 0,Y 545.093,Z 981.452,A -85,B 0,C 180,E1 3523.575,E2 3523.575} C_VEL
LIN {X 0,Y 545.719,Z 960.783,A -85,B 0,C 180,E1 3527.525,E2 3527.525} C_VEL
LIN {X 0,Y 546.883,Z 934.717,A -85,B 0,C 180,E1 3531.222,E2 3531.222} C_VEL
LIN {X 0,Y 548.374,Z 904.273,A -85,B 0,C 180,E1 3534.494,E2 3534.494} C_VEL
LIN {X 0,Y 550,Z 870.974,A -85,B 0,C 180,E1 3537.21,E2 3537.21} C_VEL
LIN {X 0,Y 551.703,Z 835.098,A -85,B 0,C 180,E1 3539.371,E2 3539.371} C_VEL
LIN {X 0,Y 553.042,Z 797.202,A -85,B 0,C 180,E1 3540.963,E2 3540.963} C_VEL
LIN {X 0,Y 554.093,Z 758.938,A -85,B 0,C 180,E1 3541.929,E2 3541.929} C_VEL
LIN {X 0,Y 553.76,Z 706.305,A -85,B 0,C 180,E1 3542.763,E2 3542.763} C_VEL
LIN {X 0,Y 544.246,Z 685.03,A -85,B 0,C 180,E1 3543.783,E2 3543.783} C_VEL
LIN {X 0,Y 543.908,Z 685.03,A -85,B 0,C 180,E1 3549.656,E2 3549.656} C_VEL
LIN {X 0,Y 544.041,Z 685.03,A -85,B 0,C 180,E1 3556.157,E2 3556.157} C_VEL
LIN {X 0,Y 544.099,Z 685.03,A -85,B 0,C 180,E1 3562.399,E2 3562.399} C_VEL
LIN {X 0,Y 543.987,Z 685.03,A -85,B 0,C 180,E1 3568.192,E2 3568.192} C_VEL
LIN {X 0,Y 544.039,Z 685.03,A -85,B 0,C 180,E1 3573.652,E2 3573.652} C_VEL
LIN {X 0,Y 544.167,Z 685.03,A -85,B 0,C 180,E1 3578.867,E2 3578.867} C_VEL
LIN {X 0,Y 544.251,Z 685.473,A -85,B 0,C 180,E1 3582.948,E2 3582.948} C_VEL
LIN {X 0,Y 547.36,Z 699.357,A -85,B 0,C 180,E1 3583.247,E2 3583.247} C_VEL
LIN {X 0,Y 547.11,Z 743.77,A -85,B 0,C 180,E1 3583.987,E2 3583.987} C_VEL
LIN {X 0,Y 546.648,Z 771.809,A -85,B 0,C 180,E1 3585.073,E2 3585.073} C_VEL
LIN {X 0,Y 545.932,Z 798.592,A -85,B 0,C 180,E1 3586.816,E2 3586.816} C_VEL
LIN {X 0,Y 545.453,Z 820.754,A -85,B 0,C 180,E1 3588.986,E2 3588.986} C_VEL
LIN {X 0,Y 545.027,Z 838.976,A -85,B 0,C 180,E1 3591.639,E2 3591.639} C_VEL
LIN {X 0,Y 544.832,Z 851.382,A -85,B 0,C 180,E1 3594.434,E2 3594.434} C_VEL
LIN {X 0,Y 544.795,Z 858.836,A -85,B 0,C 180,E1 3597.615,E2 3597.615} C_VEL
LIN {X 0,Y 544.687,Z 860.43,A -85,B 0,C 180,E1 3599.996,E2 3599.996} C_VEL
LIN {X 0,Y 544.77,Z 857.456,A -85,B 0,C 180,E1 3603.172,E2 3603.172} C_VEL
LIN {X 0,Y 544.806,Z 849.626,A -85,B 0,C 180,E1 3605.958,E2 3605.958} C_VEL
LIN {X 0,Y 545.074,Z 836.196,A -85,B 0,C 180,E1 3608.754,E2 3608.754} C_VEL
LIN {X 0,Y 545.494,Z 818.756,A -85,B 0,C 180,E1 3611.161,E2 3611.161} C_VEL
LIN {X 0,Y 546.054,Z 794.96,A -85,B 0,C 180,E1 3613.377,E2 3613.377} C_VEL
LIN {X 0,Y 546.659,Z 769.968,A -85,B 0,C 180,E1 3614.932,E2 3614.932} C_VEL
LIN {X 0,Y 547.206,Z 740.663,A -85,B 0,C 180,E1 3616.003,E2 3616.003} C_VEL
LIN {X 0,Y 546.487,Z 694.176,A -85,B 0,C 180,E1 3616.76,E2 3616.76} C_VEL
LIN {X 0,Y 544.264,Z 685.03,A -85,B 0,C 180,E1 3616.982,E2 3616.982} C_VEL
LIN {X 0,Y 544.07,Z 685.03,A -85,B 0,C 180,E1 3622.843,E2 3622.843} C_VEL
LIN {X 0,Y 543.963,Z 685.03,A -85,B 0,C 180,E1 3628.131,E2 3628.131} C_VEL
LIN {X 0,Y 543.924,Z 685.03,A -85,B 0,C 180,E1 3633.693,E2 3633.693} C_VEL
LIN {X 0,Y 544.095,Z 685.03,A -85,B 0,C 180,E1 3639.046,E2 3639.046} C_VEL
LIN {X 0,Y 543.939,Z 685.03,A -85,B 0,C 180,E1 3643.902,E2 3643.902} C_VEL
LIN {X 0,Y 544.044,Z 685.03,A -85,B 0,C 180,E1 3648.484,E2 3648.484} C_VEL
LIN {X 0,Y 543.969,Z 685.03,A -85,B 0,C 180,E1 3654.365,E2 3654.365} C_VEL
LIN {X 0,Y 544.03,Z 685.03,A -85,B 0,C 180,E1 3660.043,E2 3660.043} C_VEL
LIN {X 0,Y 544.137,Z 685.03,A -85,B 0,C 180,E1 3665.415,E2 3665.415} C_VEL
LIN {X 0,Y 544.102,Z 685.198,A -85,B 0,C 180,E1 3667.295,E2 3667.295} C_VEL
LIN {X 0,Y 549.105,Z 704.905,A -85,B 0,C 180,E1 3668.021,E2 3668.021} C_VEL
LIN {X 0,Y 548.252,Z 737.384,A -85,B 0,C 180,E1 3669.336,E2 3669.336} C_VEL
LIN {X 0,Y 547.194,Z 768.783,A -85,B 0,C 180,E1 3671.298,E2 3671.298} C_VEL
LIN {X 0,Y 546.194,Z 796.268,A -85,B 0,C 180,E1 3673.753,E2 3673.753} C_VEL
LIN {X 0,Y 545.449,Z 819.23,A -85,B 0,C 180,E1 3676.6,E2 3676.6} C_VEL
LIN {X 0,Y 544.972,Z 837.706,A -85,B 0,C 180,E1 3679.832,E2 3679.832} C_VEL
LIN {X 0,Y 544.714,Z 850.706,A -85,B 0,C 180,E1 3683.236,E2 3683.236} C_VEL
LIN {X 0,Y 544.647,Z 858.389,A -85,B 0,C 180,E1 3686.821,E2 3686.821} C_VEL
LIN {X 0,Y 544.582,Z 860.497,A -85,B 0,C 180,E1 3689.998,E2 3689.998} C_VEL
LIN {X 0,Y 544.655,Z 858.261,A -85,B 0,C 180,E1 3693.174,E2 3693.174} C_VEL
LIN {X 0,Y 544.753,Z 850.466,A -85,B 0,C 180,E1 3696.759,E2 3696.759} C_VEL
LIN {X 0,Y 544.983,Z 837.275,A -85,B 0,C 180,E1 3700.168,E2 3700.168} C_VEL
LIN {X 0,Y 545.478,Z 818.633,A -85,B 0,C 180,E1 3703.395,E2 3703.395} C_VEL
LIN {X 0,Y 546.232,Z 795.481,A -85,B 0,C 180,E1 3706.241,E2 3706.241} C_VEL
LIN {X 0,Y 547.225,Z 767.678,A -85,B 0,C 180,E1 3708.696,E2 3708.696} C_VEL
LIN {X 0,Y 548.201,Z 737.157,A -85,B 0,C 180,E1 3710.587,E2 3710.587} C_VEL
LIN {X 0,Y 549.141,Z 703.557,A -85,B 0,C 180,E1 3711.929,E2 3711.929} C_VEL
LIN {X 0,Y 544.307,Z 685.03,A -85,B 0,C 180,E1 3712.693,E2 3712.693} C_VEL
LIN {X 0,Y 544.08,Z 685.03,A -85,B 0,C 180,E1 3718.13,E2 3718.13} C_VEL
LIN {X 0,Y 544.063,Z 685.03,A -85,B 0,C 180,E1 3723.701,E2 3723.701} C_VEL
LIN {X 0,Y 543.915,Z 685.03,A -85,B 0,C 180,E1 3729.649,E2 3729.649} C_VEL
LIN {X 0,Y 543.978,Z 685.03,A -85,B 0,C 180,E1 3736.157,E2 3736.157} C_VEL
LIN {X 0,Y 544.076,Z 685.03,A -85,B 0,C 180,E1 3742.406,E2 3742.406} C_VEL
LIN {X 0,Y 544.024,Z 685.03,A -85,B 0,C 180,E1 3748.203,E2 3748.203} C_VEL
LIN {X 0,Y 544.072,Z 685.03,A -85,B 0,C 180,E1 3753.662,E2 3753.662} C_VEL
LIN {X 0,Y 544.203,Z 685.03,A -85,B 0,C 180,E1 3758.876,E2 3758.876} C_VEL
LIN {X 0,Y 544.286,Z 685.03,A -85,B 0,C 180,E1 3763.909,E2 3763.909} C_VEL
LIN {X 0,Y 544.271,Z 685.03,A -85,B 0,C 180,E1 3768.814,E2 3768.814} C_VEL
LIN {X 0,Y 544.319,Z 685.03,A -85,B 0,C 180,E1 3773.637,E2 3773.637} C_VEL
LIN {X 0,Y 544.292,Z 685.03,A -85,B 0,C 180,E1 3778.415,E2 3778.415} C_VEL
LIN {X 0,Y 544.337,Z 685.03,A -85,B 0,C 180,E1 3783.182,E2 3783.182} C_VEL
LIN {X 0,Y 544.237,Z 685.03,A -85,B 0,C 180,E1 3787.972,E2 3787.972} C_VEL
LIN {X 0,Y 544.188,Z 685.03,A -85,B 0,C 180,E1 3792.819,E2 3792.819} C_VEL
LIN {X 0,Y 544.17,Z 685.03,A -85,B 0,C 180,E1 3797.762,E2 3797.762} C_VEL
LIN {X 0,Y 544.025,Z 685.03,A -85,B 0,C 180,E1 3803.139,E2 3803.139} C_VEL
LIN {X 0,Y 540.11,Z 685.03,A -85,B 0,C 180,E1 3804.942,E2 3804.942} C_VEL
LIN {X 0,Y 536.061,Z 685.03,A -85,B 0,C 180,E1 3806.771,E2 3806.771} C_VEL
LIN {X 0,Y 536.005,Z 685.03,A -85,B 0,C 180,E1 3812.373,E2 3812.373} C_VEL
LIN {X 0,Y 536.142,Z 685.03,A -85,B 0,C 180,E1 3818.259,E2 3818.259} C_VEL
LIN {X 0,Y 535.992,Z 685.03,A -85,B 0,C 180,E1 3824.736,E2 3824.736} C_VEL
LIN {X 0,Y 535.964,Z 685.03,A -85,B 0,C 180,E1 3829.643,E2 3829.643} C_VEL
LIN {X 0,Y 536.073,Z 685.329,A -85,B 0,C 180,E1 3834.206,E2 3834.206} C_VEL
LIN {X 0,Y 537.549,Z 689.548,A -85,B 0,C 180,E1 3834.913,E2 3834.913} C_VEL
LIN {X 0,Y 539.265,Z 692.825,A -85,B 0,C 180,E1 3836.029,E2 3836.029} C_VEL
LIN {X 0,Y 547.42,Z 709.655,A -85,B 0,C 180,E1 3836.861,E2 3836.861} C_VEL
LIN {X 0,Y 546.908,Z 775.122,A -85,B 0,C 180,E1 3837.965,E2 3837.965} C_VEL
LIN {X 0,Y 545.667,Z 814.026,A -85,B 0,C 180,E1 3839.237,E2 3839.237} C_VEL
LIN {X 0,Y 543.905,Z 851.1,A -85,B 0,C 180,E1 3841.096,E2 3841.096} C_VEL
LIN {X 0,Y 541.979,Z 887.409,A -85,B 0,C 180,E1 3843.659,E2 3843.659} C_VEL
LIN {X 0,Y 540.031,Z 920.098,A -85,B 0,C 180,E1 3846.755,E2 3846.755} C_VEL
LIN {X 0,Y 538.495,Z 948.751,A -85,B 0,C 180,E1 3850.352,E2 3850.352} C_VEL
LIN {X 0,Y 537.464,Z 971.392,A -85,B 0,C 180,E1 3854.114,E2 3854.114} C_VEL
LIN {X 0,Y 536.977,Z 988.017,A -85,B 0,C 180,E1 3857.835,E2 3857.835} C_VEL
LIN {X 0,Y 536.814,Z 999.718,A -85,B 0,C 180,E1 3861.515,E2 3861.515} C_VEL
LIN {X 0,Y 536.654,Z 1006.983,A -85,B 0,C 180,E1 3865.163,E2 3865.163} C_VEL
LIN {X 0,Y 536.66,Z 1010.106,A -85,B 0,C 180,E1 3868.391,E2 3868.391} C_VEL
LIN {X 0,Y 536.797,Z 1010.103,A -85,B 0,C 180,E1 3871.613,E2 3871.613} C_VEL
LIN {X 0,Y 536.758,Z 1005.743,A -85,B 0,C 180,E1 3875.65,E2 3875.65} C_VEL
LIN {X 0,Y 536.836,Z 996.319,A -85,B 0,C 180,E1 3879.713,E2 3879.713} C_VEL
LIN {X 0,Y 537.258,Z 980.759,A -85,B 0,C 180,E1 3883.937,E2 3883.937} C_VEL
LIN {X 0,Y 538.06,Z 959.647,A -85,B 0,C 180,E1 3887.972,E2 3887.972} C_VEL
LIN {X 0,Y 539.352,Z 933.555,A -85,B 0,C 180,E1 3891.68,E2 3891.68} C_VEL
LIN {X 0,Y 541.062,Z 902.185,A -85,B 0,C 180,E1 3895.05,E2 3895.05} C_VEL
LIN {X 0,Y 542.984,Z 867.312,A -85,B 0,C 180,E1 3897.864,E2 3897.864} C_VEL
LIN {X 0,Y 544.918,Z 829.982,A -85,B 0,C 180,E1 3900.05,E2 3900.05} C_VEL
LIN {X 0,Y 546.448,Z 790.371,A -85,B 0,C 180,E1 3901.619,E2 3901.619} C_VEL
LIN {X 0,Y 547.494,Z 750.742,A -85,B 0,C 180,E1 3902.505,E2 3902.505} C_VEL
LIN {X 0,Y 547.181,Z 709.052,A -85,B 0,C 180,E1 3903.165,E2 3903.165} C_VEL
LIN {X 0,Y 539.153,Z 692.041,A -85,B 0,C 180,E1 3904.045,E2 3904.045} C_VEL
LIN {X 0,Y 536.787,Z 688.309,A -85,B 0,C 180,E1 3905.39,E2 3905.39} C_VEL
LIN {X 0,Y 536.033,Z 685.03,A -85,B 0,C 180,E1 3905.991,E2 3905.991} C_VEL
LIN {X 0,Y 535.973,Z 685.03,A -85,B 0,C 180,E1 3912.515,E2 3912.515} C_VEL
LIN {X 0,Y 536.067,Z 685.03,A -85,B 0,C 180,E1 3917.5,E2 3917.5} C_VEL
LIN {X 0,Y 536.115,Z 685.03,A -85,B 0,C 180,E1 3923.765,E2 3923.765} C_VEL
LIN {X 0,Y 536.069,Z 685.03,A -85,B 0,C 180,E1 3929.555,E2 3929.555} C_VEL
LIN {X 0,Y 536.129,Z 685.03,A -85,B 0,C 180,E1 3935.025,E2 3935.025} C_VEL
LIN {X 0,Y 536.256,Z 685.03,A -85,B 0,C 180,E1 3940.263,E2 3940.263} C_VEL
LIN {X 0,Y 536.316,Z 685.388,A -85,B 0,C 180,E1 3942.613,E2 3942.613} C_VEL
LIN {X 0,Y 539.869,Z 701.895,A -85,B 0,C 180,E1 3943.013,E2 3943.013} C_VEL
LIN {X 0,Y 539.569,Z 744.715,A -85,B 0,C 180,E1 3943.757,E2 3943.757} C_VEL
LIN {X 0,Y 539.039,Z 772.228,A -85,B 0,C 180,E1 3944.857,E2 3944.857} C_VEL
LIN {X 0,Y 538.162,Z 799.858,A -85,B 0,C 180,E1 3946.725,E2 3946.725} C_VEL
LIN {X 0,Y 537.645,Z 821.211,A -85,B 0,C 180,E1 3948.884,E2 3948.884} C_VEL
LIN {X 0,Y 537.185,Z 838.962,A -85,B 0,C 180,E1 3951.516,E2 3951.516} C_VEL
LIN {X 0,Y 536.94,Z 851.382,A -85,B 0,C 180,E1 3954.352,E2 3954.352} C_VEL
LIN {X 0,Y 536.908,Z 858.829,A -85,B 0,C 180,E1 3957.58,E2 3957.58} C_VEL
LIN {X 0,Y 536.811,Z 860.421,A -85,B 0,C 180,E1 3959.996,E2 3959.996} C_VEL
LIN {X 0,Y 536.878,Z 857.46,A -85,B 0,C 180,E1 3963.219,E2 3963.219} C_VEL
LIN {X 0,Y 536.925,Z 849.62,A -85,B 0,C 180,E1 3966.046,E2 3966.046} C_VEL
LIN {X 0,Y 537.203,Z 835.029,A -85,B 0,C 180,E1 3969.087,E2 3969.087} C_VEL
LIN {X 0,Y 537.729,Z 816.887,A -85,B 0,C 180,E1 3971.529,E2 3971.529} C_VEL
LIN {X 0,Y 538.379,Z 793.663,A -85,B 0,C 180,E1 3973.675,E2 3973.675} C_VEL
LIN {X 0,Y 539.125,Z 767.236,A -85,B 0,C 180,E1 3975.283,E2 3975.283} C_VEL
LIN {X 0,Y 539.7,Z 738.773,A -85,B 0,C 180,E1 3976.296,E2 3976.296} C_VEL
LIN {X 0,Y 539.052,Z 695.588,A -85,B 0,C 180,E1 3977.008,E2 3977.008} C_VEL
LIN {X 0,Y 536.327,Z 685.03,A -85,B 0,C 180,E1 3977.324,E2 3977.324} C_VEL
LIN {X 0,Y 536.153,Z 685.03,A -85,B 0,C 180,E1 3983.199,E2 3983.199} C_VEL
LIN {X 0,Y 535.993,Z 685.03,A -85,B 0,C 180,E1 3989.209,E2 3989.209} C_VEL
LIN {X 0,Y 536.055,Z 685.03,A -85,B 0,C 180,E1 3995.27,E2 3995.27} C_VEL
LIN {X 0,Y 536.032,Z 685.03,A -85,B 0,C 180,E1 4000.521,E2 4000.521} C_VEL
LIN {X 0,Y 536.029,Z 685.03,A -85,B 0,C 180,E1 4007.039,E2 4007.039} C_VEL
LIN {X 0,Y 536.124,Z 685.03,A -85,B 0,C 180,E1 4011.996,E2 4011.996} C_VEL
LIN {X 0,Y 536.043,Z 685.03,A -85,B 0,C 180,E1 4017.661,E2 4017.661} C_VEL
LIN {X 0,Y 536.172,Z 685.03,A -85,B 0,C 180,E1 4023.233,E2 4023.233} C_VEL
LIN {X 0,Y 536.226,Z 685.698,A -85,B 0,C 180,E1 4026.932,E2 4026.932} C_VEL
LIN {X 0,Y 541.721,Z 706.7,A -85,B 0,C 180,E1 4027.767,E2 4027.767} C_VEL
LIN {X 0,Y 540.738,Z 739.465,A -85,B 0,C 180,E1 4029.145,E2 4029.145} C_VEL
LIN {X 0,Y 539.594,Z 770.128,A -85,B 0,C 180,E1 4031.131,E2 4031.131} C_VEL
LIN {X 0,Y 538.443,Z 798.144,A -85,B 0,C 180,E1 4033.721,E2 4033.721} C_VEL
LIN {X 0,Y 537.622,Z 820.584,A -85,B 0,C 180,E1 4036.608,E2 4036.608} C_VEL
LIN {X 0,Y 537.109,Z 838.539,A -85,B 0,C 180,E1 4039.86,E2 4039.86} C_VEL
LIN {X 0,Y 536.83,Z 850.705,A -85,B 0,C 180,E1 4043.136,E2 4043.136} C_VEL
LIN {X 0,Y 536.753,Z 858.388,A -85,B 0,C 180,E1 4046.774,E2 4046.774} C_VEL
LIN {X 0,Y 536.705,Z 860.497,A -85,B 0,C 180,E1 4049.998,E2 4049.998} C_VEL
LIN {X 0,Y 536.761,Z 858.262,A -85,B 0,C 180,E1 4053.221,E2 4053.221} C_VEL
LIN {X 0,Y 536.863,Z 850.469,A -85,B 0,C 180,E1 4056.859,E2 4056.859} C_VEL
LIN {X 0,Y 537.157,Z 836.944,A -85,B 0,C 180,E1 4060.389,E2 4060.389} C_VEL
LIN {X 0,Y 537.689,Z 818.635,A -85,B 0,C 180,E1 4063.592,E2 4063.592} C_VEL
LIN {X 0,Y 538.541,Z 795.502,A -85,B 0,C 180,E1 4066.478,E2 4066.478} C_VEL
LIN {X 0,Y 539.654,Z 767.684,A -85,B 0,C 180,E1 4068.968,E2 4068.968} C_VEL
LIN {X 0,Y 540.765,Z 737.164,A -85,B 0,C 180,E1 4070.883,E2 4070.883} C_VEL
LIN {X 0,Y 541.776,Z 705.121,A -85,B 0,C 180,E1 4072.195,E2 4072.195} C_VEL
LIN {X 0,Y 536.344,Z 685.03,A -85,B 0,C 180,E1 4073.012,E2 4073.012} C_VEL
LIN {X 0,Y 536.099,Z 685.03,A -85,B 0,C 180,E1 4079.256,E2 4079.256} C_VEL
LIN {X 0,Y 536.088,Z 685.03,A -85,B 0,C 180,E1 4084.26,E2 4084.26} C_VEL
LIN {X 0,Y 535.955,Z 685.03,A -85,B 0,C 180,E1 4090.358,E2 4090.358} C_VEL
LIN {X 0,Y 535.962,Z 685.03,A -85,B 0,C 180,E1 4095.271,E2 4095.271} C_VEL
LIN {X 0,Y 536.126,Z 685.03,A -85,B 0,C 180,E1 4101.749,E2 4101.749} C_VEL
LIN {X 0,Y 536.077,Z 685.03,A -85,B 0,C 180,E1 4107.675,E2 4107.675} C_VEL
LIN {X 0,Y 536.137,Z 685.03,A -85,B 0,C 180,E1 4113.241,E2 4113.241} C_VEL
LIN {X 0,Y 536.236,Z 685.03,A -85,B 0,C 180,E1 4118.547,E2 4118.547} C_VEL
